LIN {X 0,Y 523.406,Z 267.821,A -85,B 0,C 180,E1 -4877.989,E2 -4877.989} C_VEL
LIN {X 0,Y 523.415,Z 265.36,A -85,B 0,C 180,E1 -4880.433,E2 -4880.433} C_VEL
LIN {X 0,Y 523.474,Z 262.881,A -85,B 0,C 180,E1 -4882.914,E2 -4882.914} C_VEL
LIN {X 0,Y 523.555,Z 259.879,A -85,B 0,C 180,E1 -4885.922,E2 -4885.922} C_VEL
LIN {X 0,Y 523.518,Z 256.912,A -85,B 0,C 180,E1 -4888.9,E2 -4888.9} C_VEL
LIN {X 0,Y 523.561,Z 255.036,A -85,B 0,C 180,E1 -4890.784,E2 -4890.784} C_VEL
LIN {X 0,Y 523.861,Z 254.859,A -85,B 0,C 180,E1 -4893.718,E2 -4893.718} C_VEL
LIN {X 0,Y 523.902,Z 254.849,A -85,B 0,C 180,E1 -4896.4,E2 -4896.4} C_VEL
LIN {X 0,Y 523.923,Z 254.848,A -85,B 0,C 180,E1 -4899.085,E2 -4899.085} C_VEL
LIN {X 0,Y 523.941,Z 254.846,A -85,B 0,C 180,E1 -4901.106,E2 -4901.106} C_VEL
LIN {X 0,Y 523.299,Z 254.928,A -85,B 0,C 180,E1 -4901.746,E2 -4901.746} C_VEL
LIN {X 0,Y 520.427,Z 255.284,A -85,B 0,C 180,E1 -4902.786,E2 -4902.786} C_VEL
LIN {X 0,Y 517.987,Z 255.586,A -85,B 0,C 180,E1 -4903.623,E2 -4903.623} C_VEL
LIN {X 0,Y 516.948,Z 255.716,A -85,B 0,C 180,E1 -4904.27,E2 -4904.27} C_VEL
LIN {X 0,Y 516.869,Z 255.723,A -85,B 0,C 180,E1 -4904.489,E2 -4904.489} C_VEL
LIN {X 0,Y 516.888,Z 255.725,A -85,B 0,C 180,E1 -4907.242,E2 -4907.242} C_VEL
LIN {X 0,Y 516.888,Z 255.725,A -85,B 0,C 180,E1 -4909.59,E2 -4909.59} C_VEL
LIN {X 0,Y 516.865,Z 255.729,A -85,B 0,C 180,E1 -4912.274,E2 -4912.274} C_VEL
LIN {X 0,Y 516.883,Z 255.728,A -85,B 0,C 180,E1 -4915.175,E2 -4915.175} C_VEL
LIN {X 0,Y 516.876,Z 255.725,A -85,B 0,C 180,E1 -4917.975,E2 -4917.975} C_VEL
LIN {X 0,Y 516.926,Z 255.719,A -85,B 0,C 180,E1 -4920.696,E2 -4920.696} C_VEL
LIN {X 0,Y 516.909,Z 255.722,A -85,B 0,C 180,E1 -4923.341,E2 -4923.341} C_VEL
LIN {X 0,Y 516.888,Z 255.726,A -85,B 0,C 180,E1 -4925.927,E2 -4925.927} C_VEL
LIN {X 0,Y 516.916,Z 255.722,A -85,B 0,C 180,E1 -4929.299,E2 -4929.299} C_VEL
LIN {X 0,Y 516.9,Z 255.723,A -85,B 0,C 180,E1 -4932.595,E2 -4932.595} C_VEL
LIN {X 0,Y 516.946,Z 255.72,A -85,B 0,C 180,E1 -4935.03,E2 -4935.03} C_VEL
LIN {X 0,Y 516.97,Z 255.718,A -85,B 0,C 180,E1 -4938.234,E2 -4938.234} C_VEL
LIN {X 0,Y 516.969,Z 255.717,A -85,B 0,C 180,E1 -4941.4,E2 -4941.4} C_VEL
LIN {X 0,Y 516.991,Z 255.712,A -85,B 0,C 180,E1 -4944.54,E2 -4944.54} C_VEL
LIN {X 0,Y 517.087,Z 255.701,A -85,B 0,C 180,E1 -4947.663,E2 -4947.663} C_VEL
LIN {X 0,Y 517.091,Z 255.699,A -85,B 0,C 180,E1 -4950.779,E2 -4950.779} C_VEL
LIN {X 0,Y 516.985,Z 255.713,A -85,B 0,C 180,E1 -4953.117,E2 -4953.117} C_VEL
LIN {X 0,Y 516.997,Z 255.713,A -85,B 0,C 180,E1 -4956.243,E2 -4956.243} C_VEL
LIN {X 0,Y 516.942,Z 255.719,A -85,B 0,C 180,E1 -4959.39,E2 -4959.39} C_VEL
LIN {X 0,Y 516.956,Z 255.715,A -85,B 0,C 180,E1 -4961.807,E2 -4961.807} C_VEL
LIN {X 0,Y 516.943,Z 255.717,A -85,B 0,C 180,E1 -4965.144,E2 -4965.144} C_VEL
LIN {X 0,Y 516.92,Z 255.721,A -85,B 0,C 180,E1 -4968.223,E2 -4968.223} C_VEL
LIN {X 0,Y 516.916,Z 255.72,A -85,B 0,C 180,E1 -4970.702,E2 -4970.702} C_VEL
LIN {X 0,Y 516.905,Z 255.721,A -85,B 0,C 180,E1 -4974.073,E2 -4974.073} C_VEL
LIN {X 0,Y 516.926,Z 255.72,A -85,B 0,C 180,E1 -4976.658,E2 -4976.658} C_VEL
LIN {X 0,Y 516.91,Z 255.723,A -85,B 0,C 180,E1 -4979.523,E2 -4979.523} C_VEL
LIN {X 0,Y 516.9,Z 255.726,A -85,B 0,C 180,E1 -4982.543,E2 -4982.543} C_VEL
LIN {X 0,Y 516.866,Z 255.731,A -85,B 0,C 180,E1 -4985.329,E2 -4985.329} C_VEL
LIN {X 0,Y 516.882,Z 255.725,A -85,B 0,C 180,E1 -4987.943,E2 -4987.943} C_VEL
LIN {X 0,Y 516.864,Z 255.727,A -85,B 0,C 180,E1 -4990.744,E2 -4990.744} C_VEL
LIN {X 0,Y 516.884,Z 255.723,A -85,B 0,C 180,E1 -4993.904,E2 -4993.904} C_VEL
LIN {X 0,Y 516.887,Z 255.727,A -85,B 0,C 180,E1 -4996.107,E2 -4996.107} C_VEL
LIN {X 0,Y 516.917,Z 255.72,A -85,B 0,C 180,E1 -4998.399,E2 -4998.399} C_VEL
LIN {X 0,Y 516.883,Z 255.724,A -85,B 0,C 180,E1 -5001.284,E2 -5001.284} C_VEL
LIN {X 0,Y 516.875,Z 255.726,A -85,B 0,C 180,E1 -5004.22,E2 -5004.22} C_VEL
LIN {X 0,Y 516.886,Z 255.725,A -85,B 0,C 180,E1 -5007.052,E2 -5007.052} C_VEL
LIN {X 0,Y 516.897,Z 255.725,A -85,B 0,C 180,E1 -5009.796,E2 -5009.796} C_VEL
LIN {X 0,Y 516.928,Z 255.72,A -85,B 0,C 180,E1 -5012.467,E2 -5012.467} C_VEL
LIN {X 0,Y 516.89,Z 255.725,A -85,B 0,C 180,E1 -5015.642,E2 -5015.642} C_VEL
LIN {X 0,Y 516.89,Z 255.724,A -85,B 0,C 180,E1 -5018.462,E2 -5018.462} C_VEL
LIN {X 0,Y 516.896,Z 255.722,A -85,B 0,C 180,E1 -5020.954,E2 -5020.954} C_VEL
LIN {X 0,Y 516.907,Z 255.724,A -85,B 0,C 180,E1 -5023.41,E2 -5023.41} C_VEL
LIN {X 0,Y 516.886,Z 255.724,A -85,B 0,C 180,E1 -5025.833,E2 -5025.833} C_VEL
LIN {X 0,Y 516.957,Z 255.715,A -85,B 0,C 180,E1 -5029.028,E2 -5029.028} C_VEL
LIN {X 0,Y 516.949,Z 255.717,A -85,B 0,C 180,E1 -5032.186,E2 -5032.186} C_VEL
LIN {X 0,Y 516.991,Z 255.711,A -85,B 0,C 180,E1 -5034.539,E2 -5034.539} C_VEL
LIN {X 0,Y 517.088,Z 255.7,A -85,B 0,C 180,E1 -5037.663,E2 -5037.663} C_VEL
LIN {X 0,Y 517.09,Z 255.701,A -85,B 0,C 180,E1 -5040,E2 -5040} C_VEL
LIN {X 0,Y 517.014,Z 255.71,A -85,B 0,C 180,E1 -5043.117,E2 -5043.117} C_VEL
LIN {X 0,Y 516.992,Z 255.715,A -85,B 0,C 180,E1 -5046.243,E2 -5046.243} C_VEL
LIN {X 0,Y 516.944,Z 255.72,A -85,B 0,C 180,E1 -5049.389,E2 -5049.389} C_VEL
LIN {X 0,Y 516.957,Z 255.716,A -85,B 0,C 180,E1 -5051.807,E2 -5051.807} C_VEL
LIN {X 0,Y 516.943,Z 255.717,A -85,B 0,C 180,E1 -5055.144,E2 -5055.144} C_VEL
LIN {X 0,Y 516.921,Z 255.722,A -85,B 0,C 180,E1 -5058.222,E2 -5058.222} C_VEL
LIN {X 0,Y 516.909,Z 255.72,A -85,B 0,C 180,E1 -5060.701,E2 -5060.701} C_VEL
LIN {X 0,Y 516.893,Z 255.724,A -85,B 0,C 180,E1 -5064.073,E2 -5064.073} C_VEL
LIN {X 0,Y 516.893,Z 255.723,A -85,B 0,C 180,E1 -5066.659,E2 -5066.659} C_VEL
LIN {X 0,Y 516.889,Z 255.725,A -85,B 0,C 180,E1 -5069.518,E2 -5069.518} C_VEL
LIN {X 0,Y 516.898,Z 255.724,A -85,B 0,C 180,E1 -5072.543,E2 -5072.543} C_VEL
LIN {X 0,Y 516.863,Z 255.73,A -85,B 0,C 180,E1 -5075.328,E2 -5075.328} C_VEL
LIN {X 0,Y 516.884,Z 255.725,A -85,B 0,C 180,E1 -5077.943,E2 -5077.943} C_VEL
LIN {X 0,Y 516.863,Z 255.727,A -85,B 0,C 180,E1 -5080.743,E2 -5080.743} C_VEL
LIN {X 0,Y 516.93,Z 255.935,A -85,B 0,C 180,E1 -5083.898,E2 -5083.898} C_VEL
LIN {X 0,Y 518.179,Z 262.543,A -85,B 0,C 180,E1 -5087.087,E2 -5087.087} C_VEL
LIN {X 0,Y 518.507,Z 266.609,A -85,B 0,C 180,E1 -5088.899,E2 -5088.899} C_VEL
LIN {X 0,Y 518.31,Z 272.634,A -85,B 0,C 180,E1 -5091.41,E2 -5091.41} C_VEL
LIN {X 0,Y 518.056,Z 279.916,A -85,B 0,C 180,E1 -5094.314,E2 -5094.314} C_VEL
LIN {X 0,Y 517.764,Z 287.94,A -85,B 0,C 180,E1 -5097.306,E2 -5097.306} C_VEL
LIN {X 0,Y 517.585,Z 296.354,A -85,B 0,C 180,E1 -5100.345,E2 -5100.345} C_VEL
LIN {X 0,Y 517.316,Z 305.881,A -85,B 0,C 180,E1 -5103.72,E2 -5103.72} C_VEL
LIN {X 0,Y 517.036,Z 314.769,A -85,B 0,C 180,E1 -5106.784,E2 -5106.784} C_VEL
LIN {X 0,Y 516.833,Z 323.591,A -85,B 0,C 180,E1 -5109.764,E2 -5109.764} C_VEL
LIN {X 0,Y 516.808,Z 325.424,A -85,B 0,C 180,E1 -5110.376,E2 -5110.376} C_VEL
LIN {X 0,Y 520.665,Z 341.342,A -85,B 0,C 180,E1 -5110.82,E2 -5110.82} C_VEL
LIN {X 0,Y 520.389,Z 357.008,A -85,B 0,C 180,E1 -5111.264,E2 -5111.264} C_VEL
LIN {X 0,Y 520.036,Z 371.091,A -85,B 0,C 180,E1 -5111.817,E2 -5111.817} C_VEL
LIN {X 0,Y 519.543,Z 384.386,A -85,B 0,C 180,E1 -5112.483,E2 -5112.483} C_VEL
LIN {X 0,Y 518.999,Z 398.66,A -85,B 0,C 180,E1 -5113.377,E2 -5113.377} C_VEL
LIN {X 0,Y 518.459,Z 411.744,A -85,B 0,C 180,E1 -5114.386,E2 -5114.386} C_VEL
LIN {X 0,Y 517.949,Z 423.365,A -85,B 0,C 180,E1 -5115.462,E2 -5115.462} C_VEL
LIN {X 0,Y 517.566,Z 434.168,A -85,B 0,C 180,E1 -5116.653,E2 -5116.653} C_VEL
LIN {X 0,Y 517.117,Z 444.315,A -85,B 0,C 180,E1 -5117.983,E2 -5117.983} C_VEL
LIN {X 0,Y 516.889,Z 453.439,A -85,B 0,C 180,E1 -5119.423,E2 -5119.423} C_VEL
LIN {X 0,Y 516.581,Z 461.637,A -85,B 0,C 180,E1 -5120.999,E2 -5120.999} C_VEL
LIN {X 0,Y 516.428,Z 468.204,A -85,B 0,C 180,E1 -5122.572,E2 -5122.572} C_VEL
LIN {X 0,Y 516.378,Z 473.338,A -85,B 0,C 180,E1 -5124.141,E2 -5124.141} C_VEL
LIN {X 0,Y 516.239,Z 476.297,A -85,B 0,C 180,E1 -5125.315,E2 -5125.315} C_VEL
LIN {X 0,Y 516.271,Z 479.191,A -85,B 0,C 180,E1 -5126.879,E2 -5126.879} C_VEL
LIN {X 0,Y 516.189,Z 480.915,A -85,B 0,C 180,E1 -5128.44,E2 -5128.44} C_VEL
LIN {X 0,Y 516.151,Z 481.5,A -85,B 0,C 180,E1 -5130,E2 -5130} C_VEL
LIN {X 0,Y 516.189,Z 480.912,A -85,B 0,C 180,E1 -5131.56,E2 -5131.56} C_VEL
LIN {X 0,Y 516.271,Z 479.185,A -85,B 0,C 180,E1 -5133.121,E2 -5133.121} C_VEL
LIN {X 0,Y 516.239,Z 476.294,A -85,B 0,C 180,E1 -5134.685,E2 -5134.685} C_VEL
LIN {X 0,Y 516.376,Z 472.164,A -85,B 0,C 180,E1 -5136.251,E2 -5136.251} C_VEL
LIN {X 0,Y 516.463,Z 466.693,A -85,B 0,C 180,E1 -5137.821,E2 -5137.821} C_VEL
LIN {X 0,Y 516.627,Z 459.735,A -85,B 0,C 180,E1 -5139.395,E2 -5139.395} C_VEL
LIN {X 0,Y 516.974,Z 451.086,A -85,B 0,C 180,E1 -5140.972,E2 -5140.972} C_VEL
LIN {X 0,Y 517.204,Z 442.012,A -85,B 0,C 180,E1 -5142.338,E2 -5142.338} C_VEL
LIN {X 0,Y 517.611,Z 432.477,A -85,B 0,C 180,E1 -5143.546,E2 -5143.546} C_VEL
LIN {X 0,Y 518.043,Z 421.354,A -85,B 0,C 180,E1 -5144.736,E2 -5144.736} C_VEL
LIN {X 0,Y 518.503,Z 409.888,A -85,B 0,C 180,E1 -5145.77,E2 -5145.77} C_VEL
LIN {X 0,Y 519.031,Z 397.214,A -85,B 0,C 180,E1 -5146.723,E2 -5146.723} C_VEL
LIN {X 0,Y 519.558,Z 384.408,A -85,B 0,C 180,E1 -5147.516,E2 -5147.516} C_VEL
LIN {X 0,Y 520.032,Z 371.116,A -85,B 0,C 180,E1 -5148.183,E2 -5148.183} C_VEL
LIN {X 0,Y 520.461,Z 355.507,A -85,B 0,C 180,E1 -5148.785,E2 -5148.785} C_VEL
LIN {X 0,Y 520.675,Z 341.247,A -85,B 0,C 180,E1 -5149.183,E2 -5149.183} C_VEL
LIN {X 0,Y 516.802,Z 325.427,A -85,B 0,C 180,E1 -5149.623,E2 -5149.623} C_VEL
LIN {X 0,Y 516.961,Z 318.483,A -85,B 0,C 180,E1 -5151.954,E2 -5151.954} C_VEL
LIN {X 0,Y 517.153,Z 309.818,A -85,B 0,C 180,E1 -5154.916,E2 -5154.916} C_VEL
LIN {X 0,Y 517.345,Z 302.391,A -85,B 0,C 180,E1 -5157.509,E2 -5157.509} C_VEL
LIN {X 0,Y 517.567,Z 294.891,A -85,B 0,C 180,E1 -5160.16,E2 -5160.16} C_VEL
LIN {X 0,Y 517.732,Z 285.622,A -85,B 0,C 180,E1 -5163.352,E2 -5163.352} C_VEL
LIN {X 0,Y 517.912,Z 279.176,A -85,B 0,C 180,E1 -5165.698,E2 -5165.698} C_VEL
LIN {X 0,Y 518.22,Z 272.13,A -85,B 0,C 180,E1 -5168.598,E2 -5168.598} C_VEL
LIN {X 0,Y 518.476,Z 267.989,A -85,B 0,C 180,E1 -5170.616,E2 -5170.616} C_VEL
LIN {X 0,Y 518.547,Z 265.926,A -85,B 0,C 180,E1 -5171.804,E2 -5171.804} C_VEL
LIN {X 0,Y 518.255,Z 263.34,A -85,B 0,C 180,E1 -5173.758,E2 -5173.758} C_VEL
LIN {X 0,Y 517.9,Z 261.592,A -85,B 0,C 180,E1 -5175.991,E2 -5175.991} C_VEL
LIN {X 0,Y 517.599,Z 261.084,A -85,B 0,C 180,E1 -5178.314,E2 -5178.314} C_VEL
LIN {X 0,Y 517.206,Z 261.849,A -85,B 0,C 180,E1 -5181.313,E2 -5181.313} C_VEL
LIN {X 0,Y 516.978,Z 263.353,A -85,B 0,C 180,E1 -5184.228,E2 -5184.228} C_VEL
LIN {X 0,Y 516.825,Z 265.149,A -85,B 0,C 180,E1 -5187.048,E2 -5187.048} C_VEL
LIN {X 0,Y 516.727,Z 267.071,A -85,B 0,C 180,E1 -5189.786,E2 -5189.786} C_VEL
LIN {X 0,Y 516.626,Z 269.077,A -85,B 0,C 180,E1 -5192.45,E2 -5192.45} C_VEL
LIN {X 0,Y 516.508,Z 271.145,A -85,B 0,C 180,E1 -5195.051,E2 -5195.051} C_VEL
LIN {X 0,Y 516.464,Z 272.453,A -85,B 0,C 180,E1 -5196.638,E2 -5196.638} C_VEL
LIN {X 0,Y 520.318,Z 286.354,A -85,B 0,C 180,E1 -5197.076,E2 -5197.076} C_VEL
LIN {X 0,Y 520.049,Z 302.179,A -85,B 0,C 180,E1 -5197.565,E2 -5197.565} C_VEL
LIN {X 0,Y 519.665,Z 317.564,A -85,B 0,C 180,E1 -5198.219,E2 -5198.219} C_VEL
LIN {X 0,Y 519.183,Z 331.854,A -85,B 0,C 180,E1 -5199,E2 -5199} C_VEL
LIN {X 0,Y 518.738,Z 345.039,A -85,B 0,C 180,E1 -5199.892,E2 -5199.892} C_VEL
LIN {X 0,Y 518.269,Z 357.321,A -85,B 0,C 180,E1 -5200.904,E2 -5200.904} C_VEL
LIN {X 0,Y 517.822,Z 369.228,A -85,B 0,C 180,E1 -5202.082,E2 -5202.082} C_VEL
LIN {X 0,Y 517.375,Z 380.417,A -85,B 0,C 180,E1 -5203.426,E2 -5203.426} C_VEL
LIN {X 0,Y 517.06,Z 388.916,A -85,B 0,C 180,E1 -5204.64,E2 -5204.64} C_VEL
LIN {X 0,Y 516.787,Z 397.101,A -85,B 0,C 180,E1 -5206.032,E2 -5206.032} C_VEL
LIN {X 0,Y 516.568,Z 403.816,A -85,B 0,C 180,E1 -5207.427,E2 -5207.427} C_VEL
LIN {X 0,Y 516.41,Z 410.046,A -85,B 0,C 180,E1 -5209.016,E2 -5209.016} C_VEL
LIN {X 0,Y 516.275,Z 414.768,A -85,B 0,C 180,E1 -5210.599,E2 -5210.599} C_VEL
LIN {X 0,Y 516.26,Z 418.206,A -85,B 0,C 180,E1 -5212.176,E2 -5212.176} C_VEL
LIN {X 0,Y 516.295,Z 420.481,A -85,B 0,C 180,E1 -5213.748,E2 -5213.748} C_VEL
LIN {X 0,Y 516.213,Z 421.519,A -85,B 0,C 180,E1 -5215.315,E2 -5215.315} C_VEL
LIN {X 0,Y 516.278,Z 421.689,A -85,B 0,C 180,E1 -5216.097,E2 -5216.097} C_VEL
LIN {X 0,Y 516.258,Z 421.036,A -85,B 0,C 180,E1 -5217.66,E2 -5217.66} C_VEL
LIN {X 0,Y 516.16,Z 419.321,A -85,B 0,C 180,E1 -5219.22,E2 -5219.22} C_VEL
LIN {X 0,Y 516.181,Z 416.483,A -85,B 0,C 180,E1 -5220.78,E2 -5220.78} C_VEL
LIN {X 0,Y 516.314,Z 412.311,A -85,B 0,C 180,E1 -5222.341,E2 -5222.341} C_VEL
LIN {X 0,Y 516.495,Z 408.36,A -85,B 0,C 180,E1 -5223.511,E2 -5223.511} C_VEL
LIN {X 0,Y 516.663,Z 401.892,A -85,B 0,C 180,E1 -5225.073,E2 -5225.073} C_VEL
LIN {X 0,Y 516.849,Z 394.528,A -85,B 0,C 180,E1 -5226.5,E2 -5226.5} C_VEL
LIN {X 0,Y 517.127,Z 386.378,A -85,B 0,C 180,E1 -5227.811,E2 -5227.811} C_VEL
LIN {X 0,Y 517.527,Z 376.249,A -85,B 0,C 180,E1 -5229.182,E2 -5229.182} C_VEL
LIN {X 0,Y 517.917,Z 365.769,A -85,B 0,C 180,E1 -5230.358,E2 -5230.358} C_VEL
LIN {X 0,Y 518.424,Z 354.456,A -85,B 0,C 180,E1 -5231.436,E2 -5231.436} C_VEL
LIN {X 0,Y 518.943,Z 340.7,A -85,B 0,C 180,E1 -5232.515,E2 -5232.515} C_VEL
LIN {X 0,Y 519.352,Z 328.639,A -85,B 0,C 180,E1 -5233.3,E2 -5233.3} C_VEL
LIN {X 0,Y 519.838,Z 313.549,A -85,B 0,C 180,E1 -5234.085,E2 -5234.085} C_VEL
LIN {X 0,Y 520.268,Z 298.968,A -85,B 0,C 180,E1 -5234.672,E2 -5234.672} C_VEL
LIN {X 0,Y 520.386,Z 286.11,A -85,B 0,C 180,E1 -5235.065,E2 -5235.065} C_VEL
LIN {X 0,Y 516.998,Z 273.328,A -85,B 0,C 180,E1 -5235.464,E2 -5235.464} C_VEL
LIN {X 0,Y 516.35,Z 270.85,A -85,B 0,C 180,E1 -5235.555,E2 -5235.555} C_VEL
LIN {X 0,Y 516.342,Z 268.172,A -85,B 0,C 180,E1 -5238.244,E2 -5238.244} C_VEL
LIN {X 0,Y 516.353,Z 265.672,A -85,B 0,C 180,E1 -5240.725,E2 -5240.725} C_VEL
LIN {X 0,Y 516.424,Z 263.167,A -85,B 0,C 180,E1 -5243.245,E2 -5243.245} C_VEL
LIN {X 0,Y 516.487,Z 260.344,A -85,B 0,C 180,E1 -5246.092,E2 -5246.092} C_VEL
LIN {X 0,Y 516.435,Z 258.002,A -85,B 0,C 180,E1 -5248.445,E2 -5248.445} C_VEL
LIN {X 0,Y 516.461,Z 256.231,A -85,B 0,C 180,E1 -5250.232,E2 -5250.232} C_VEL
LIN {X 0,Y 516.523,Z 255.774,A -85,B 0,C 180,E1 -5251.134,E2 -5251.134} C_VEL
LIN {X 0,Y 516.82,Z 255.735,A -85,B 0,C 180,E1 -5253.951,E2 -5253.951} C_VEL
LIN {X 0,Y 516.857,Z 255.728,A -85,B 0,C 180,E1 -5256.748,E2 -5256.748} C_VEL
LIN {X 0,Y 516.886,Z 255.725,A -85,B 0,C 180,E1 -5259.721,E2 -5259.721} C_VEL
LIN {X 0,Y 516.909,Z 255.723,A -85,B 0,C 180,E1 -5261.776,E2 -5261.776} C_VEL
LIN {X 0,Y 516.869,Z 255.723,A -85,B 0,C 180,E1 -5264.489,E2 -5264.489} C_VEL
LIN {X 0,Y 516.212,Z 255.809,A -85,B 0,C 180,E1 -5265.14,E2 -5265.14} C_VEL
LIN {X 0,Y 513.347,Z 256.167,A -85,B 0,C 180,E1 -5266.196,E2 -5266.196} C_VEL
LIN {X 0,Y 510.932,Z 256.468,A -85,B 0,C 180,E1 -5267.046,E2 -5267.046} C_VEL
LIN {X 0,Y 509.917,Z 256.595,A -85,B 0,C 180,E1 -5267.704,E2 -5267.704} C_VEL
LIN {X 0,Y 509.847,Z 256.602,A -85,B 0,C 180,E1 -5267.926,E2 -5267.926} C_VEL
LIN {X 0,Y 509.848,Z 256.603,A -85,B 0,C 180,E1 -5270.647,E2 -5270.647} C_VEL
LIN {X 0,Y 509.828,Z 256.606,A -85,B 0,C 180,E1 -5273.647,E2 -5273.647} C_VEL
LIN {X 0,Y 509.845,Z 256.602,A -85,B 0,C 180,E1 -5276.538,E2 -5276.538} C_VEL
LIN {X 0,Y 509.849,Z 256.601,A -85,B 0,C 180,E1 -5279.334,E2 -5279.334} C_VEL
LIN {X 0,Y 509.895,Z 256.595,A -85,B 0,C 180,E1 -5282.054,E2 -5282.054} C_VEL
LIN {X 0,Y 509.811,Z 256.607,A -85,B 0,C 180,E1 -5284.7,E2 -5284.7} C_VEL
LIN {X 0,Y 509.83,Z 256.605,A -85,B 0,C 180,E1 -5287.458,E2 -5287.458} C_VEL
LIN {X 0,Y 509.92,Z 256.591,A -85,B 0,C 180,E1 -5289.845,E2 -5289.845} C_VEL
LIN {X 0,Y 509.872,Z 256.598,A -85,B 0,C 180,E1 -5293.174,E2 -5293.174} C_VEL
LIN {X 0,Y 509.863,Z 256.6,A -85,B 0,C 180,E1 -5295.634,E2 -5295.634} C_VEL
LIN {X 0,Y 509.916,Z 256.591,A -85,B 0,C 180,E1 -5298.875,E2 -5298.875} C_VEL
LIN {X 0,Y 509.955,Z 256.588,A -85,B 0,C 180,E1 -5302.078,E2 -5302.078} C_VEL
LIN {X 0,Y 509.946,Z 256.59,A -85,B 0,C 180,E1 -5304.464,E2 -5304.464} C_VEL
LIN {X 0,Y 510.056,Z 256.577,A -85,B 0,C 180,E1 -5307.631,E2 -5307.631} C_VEL
LIN {X 0,Y 510.06,Z 256.576,A -85,B 0,C 180,E1 -5310,E2 -5310} C_VEL
LIN {X 0,Y 510.053,Z 256.575,A -85,B 0,C 180,E1 -5312.369,E2 -5312.369} C_VEL
LIN {X 0,Y 509.979,Z 256.585,A -85,B 0,C 180,E1 -5315.536,E2 -5315.536} C_VEL
LIN {X 0,Y 509.905,Z 256.592,A -85,B 0,C 180,E1 -5318.72,E2 -5318.72} C_VEL
LIN {X 0,Y 509.908,Z 256.594,A -85,B 0,C 180,E1 -5321.932,E2 -5321.932} C_VEL
LIN {X 0,Y 509.898,Z 256.595,A -85,B 0,C 180,E1 -5325.242,E2 -5325.242} C_VEL
LIN {X 0,Y 509.865,Z 256.601,A -85,B 0,C 180,E1 -5328.484,E2 -5328.484} C_VEL
LIN {X 0,Y 509.854,Z 256.6,A -85,B 0,C 180,E1 -5331.002,E2 -5331.002} C_VEL
LIN {X 0,Y 509.867,Z 256.6,A -85,B 0,C 180,E1 -5334.426,E2 -5334.426} C_VEL
LIN {X 0,Y 509.884,Z 256.596,A -85,B 0,C 180,E1 -5337.056,E2 -5337.056} C_VEL
LIN {X 0,Y 509.86,Z 256.599,A -85,B 0,C 180,E1 -5339.751,E2 -5339.751} C_VEL
LIN {X 0,Y 509.877,Z 256.598,A -85,B 0,C 180,E1 -5342.774,E2 -5342.774} C_VEL
LIN {X 0,Y 509.826,Z 256.605,A -85,B 0,C 180,E1 -5345.578,E2 -5345.578} C_VEL
LIN {X 0,Y 509.853,Z 256.602,A -85,B 0,C 180,E1 -5348.338,E2 -5348.338} C_VEL
LIN {X 0,Y 509.812,Z 256.609,A -85,B 0,C 180,E1 -5351.43,E2 -5351.43} C_VEL
LIN {X 0,Y 509.843,Z 256.605,A -85,B 0,C 180,E1 -5354.67,E2 -5354.67} C_VEL
LIN {X 0,Y 509.838,Z 256.605,A -85,B 0,C 180,E1 -5357.51,E2 -5357.51} C_VEL
LIN {X 0,Y 509.849,Z 256.605,A -85,B 0,C 180,E1 -5360.647,E2 -5360.647} C_VEL
LIN {X 0,Y 509.829,Z 256.606,A -85,B 0,C 180,E1 -5363.647,E2 -5363.647} C_VEL
LIN {X 0,Y 509.846,Z 256.603,A -85,B 0,C 180,E1 -5366.538,E2 -5366.538} C_VEL
LIN {X 0,Y 509.85,Z 256.602,A -85,B 0,C 180,E1 -5369.334,E2 -5369.334} C_VEL
LIN {X 0,Y 509.895,Z 256.594,A -85,B 0,C 180,E1 -5372.054,E2 -5372.054} C_VEL
LIN {X 0,Y 509.829,Z 256.604,A -85,B 0,C 180,E1 -5374.701,E2 -5374.701} C_VEL
LIN {X 0,Y 509.832,Z 256.605,A -85,B 0,C 180,E1 -5377.458,E2 -5377.458} C_VEL
LIN {X 0,Y 509.92,Z 256.591,A -85,B 0,C 180,E1 -5379.845,E2 -5379.845} C_VEL
LIN {X 0,Y 509.873,Z 256.6,A -85,B 0,C 180,E1 -5383.174,E2 -5383.174} C_VEL
LIN {X 0,Y 509.858,Z 256.599,A -85,B 0,C 180,E1 -5385.634,E2 -5385.634} C_VEL
LIN {X 0,Y 509.919,Z 256.592,A -85,B 0,C 180,E1 -5388.874,E2 -5388.874} C_VEL
LIN {X 0,Y 509.914,Z 256.593,A -85,B 0,C 180,E1 -5392.078,E2 -5392.078} C_VEL
LIN {X 0,Y 509.946,Z 256.589,A -85,B 0,C 180,E1 -5394.464,E2 -5394.464} C_VEL
LIN {X 0,Y 510.057,Z 256.576,A -85,B 0,C 180,E1 -5397.631,E2 -5397.631} C_VEL
LIN {X 0,Y 510.061,Z 256.577,A -85,B 0,C 180,E1 -5400,E2 -5400} C_VEL
LIN {X 0,Y 510.059,Z 256.574,A -85,B 0,C 180,E1 -5402.369,E2 -5402.369} C_VEL
LIN {X 0,Y 509.978,Z 256.585,A -85,B 0,C 180,E1 -5405.536,E2 -5405.536} C_VEL
LIN {X 0,Y 509.89,Z 256.595,A -85,B 0,C 180,E1 -5408.72,E2 -5408.72} C_VEL
LIN {X 0,Y 509.909,Z 256.594,A -85,B 0,C 180,E1 -5411.931,E2 -5411.931} C_VEL
LIN {X 0,Y 509.899,Z 256.596,A -85,B 0,C 180,E1 -5415.241,E2 -5415.241} C_VEL
LIN {X 0,Y 509.866,Z 256.601,A -85,B 0,C 180,E1 -5418.483,E2 -5418.483} C_VEL
LIN {X 0,Y 509.85,Z 256.6,A -85,B 0,C 180,E1 -5421.002,E2 -5421.002} C_VEL
LIN {X 0,Y 509.824,Z 256.604,A -85,B 0,C 180,E1 -5423.564,E2 -5423.564} C_VEL
LIN {X 0,Y 509.878,Z 256.599,A -85,B 0,C 180,E1 -5426.37,E2 -5426.37} C_VEL
LIN {X 0,Y 509.854,Z 256.6,A -85,B 0,C 180,E1 -5429.751,E2 -5429.751} C_VEL
LIN {X 0,Y 509.873,Z 256.598,A -85,B 0,C 180,E1 -5432.773,E2 -5432.773} C_VEL
LIN {X 0,Y 509.824,Z 256.605,A -85,B 0,C 180,E1 -5435.577,E2 -5435.577} C_VEL
LIN {X 0,Y 509.853,Z 256.601,A -85,B 0,C 180,E1 -5438.338,E2 -5438.338} C_VEL
LIN {X 0,Y 509.834,Z 256.605,A -85,B 0,C 180,E1 -5441.427,E2 -5441.427} C_VEL
LIN {X 0,Y 509.841,Z 256.716,A -85,B 0,C 180,E1 -5443.424,E2 -5443.424} C_VEL
LIN {X 0,Y 511.063,Z 263.043,A -85,B 0,C 180,E1 -5446.56,E2 -5446.56} C_VEL
LIN {X 0,Y 511.51,Z 265.916,A -85,B 0,C 180,E1 -5447.897,E2 -5447.897} C_VEL
LIN {X 0,Y 511.484,Z 271.465,A -85,B 0,C 180,E1 -5450.306,E2 -5450.306} C_VEL
LIN {X 0,Y 511.202,Z 278.822,A -85,B 0,C 180,E1 -5453.319,E2 -5453.319} C_VEL
LIN {X 0,Y 510.881,Z 286.102,A -85,B 0,C 180,E1 -5456.141,E2 -5456.141} C_VEL
LIN {X 0,Y 510.607,Z 294.884,A -85,B 0,C 180,E1 -5459.385,E2 -5459.385} C_VEL
LIN {X 0,Y 510.39,Z 302.391,A -85,B 0,C 180,E1 -5462.084,E2 -5462.084} C_VEL
LIN {X 0,Y 510.157,Z 309.818,A -85,B 0,C 180,E1 -5464.719,E2 -5464.719} C_VEL
LIN {X 0,Y 509.937,Z 318.662,A -85,B 0,C 180,E1 -5467.789,E2 -5467.789} C_VEL
LIN {X 0,Y 509.769,Z 325.428,A -85,B 0,C 180,E1 -5470.095,E2 -5470.095} C_VEL
LIN {X 0,Y 513.784,Z 341.933,A -85,B 0,C 180,E1 -5470.567,E2 -5470.567} C_VEL
LIN {X 0,Y 513.969,Z 347.826,A -85,B 0,C 180,E1 -5470.73,E2 -5470.73} C_VEL
LIN {X 0,Y 513.534,Z 362.77,A -85,B 0,C 180,E1 -5471.222,E2 -5471.222} C_VEL
LIN {X 0,Y 512.994,Z 377.835,A -85,B 0,C 180,E1 -5471.891,E2 -5471.891} C_VEL
LIN {X 0,Y 512.49,Z 391.111,A -85,B 0,C 180,E1 -5472.646,E2 -5472.646} C_VEL
LIN {X 0,Y 511.947,Z 404.102,A -85,B 0,C 180,E1 -5473.552,E2 -5473.552} C_VEL
LIN {X 0,Y 511.422,Z 415.612,A -85,B 0,C 180,E1 -5474.515,E2 -5474.515} C_VEL
LIN {X 0,Y 510.888,Z 427.155,A -85,B 0,C 180,E1 -5475.663,E2 -5475.663} C_VEL
LIN {X 0,Y 510.419,Z 437.363,A -85,B 0,C 180,E1 -5476.868,E2 -5476.868} C_VEL
LIN {X 0,Y 509.987,Z 447.098,A -85,B 0,C 180,E1 -5478.234,E2 -5478.234} C_VEL
LIN {X 0,Y 509.745,Z 455.642,A -85,B 0,C 180,E1 -5479.675,E2 -5479.675} C_VEL
LIN {X 0,Y 509.482,Z 463.412,A -85,B 0,C 180,E1 -5481.272,E2 -5481.272} C_VEL
LIN {X 0,Y 509.318,Z 469.602,A -85,B 0,C 180,E1 -5482.866,E2 -5482.866} C_VEL
LIN {X 0,Y 509.284,Z 474.389,A -85,B 0,C 180,E1 -5484.457,E2 -5484.457} C_VEL
LIN {X 0,Y 509.201,Z 477.895,A -85,B 0,C 180,E1 -5486.043,E2 -5486.043} C_VEL
LIN {X 0,Y 509.158,Z 480.196,A -85,B 0,C 180,E1 -5487.627,E2 -5487.627} C_VEL
LIN {X 0,Y 509.07,Z 481.351,A -85,B 0,C 180,E1 -5489.209,E2 -5489.209} C_VEL
LIN {X 0,Y 509.07,Z 481.35,A -85,B 0,C 180,E1 -5490.791,E2 -5490.791} C_VEL
LIN {X 0,Y 509.158,Z 480.191,A -85,B 0,C 180,E1 -5492.373,E2 -5492.373} C_VEL
LIN {X 0,Y 509.201,Z 477.889,A -85,B 0,C 180,E1 -5493.957,E2 -5493.957} C_VEL
LIN {X 0,Y 509.285,Z 474.388,A -85,B 0,C 180,E1 -5495.543,E2 -5495.543} C_VEL
LIN {X 0,Y 509.32,Z 469.603,A -85,B 0,C 180,E1 -5497.134,E2 -5497.134} C_VEL
LIN {X 0,Y 509.481,Z 463.409,A -85,B 0,C 180,E1 -5498.728,E2 -5498.728} C_VEL
LIN {X 0,Y 509.745,Z 455.636,A -85,B 0,C 180,E1 -5500.325,E2 -5500.325} C_VEL
LIN {X 0,Y 510.009,Z 447.014,A -85,B 0,C 180,E1 -5501.778,E2 -5501.778} C_VEL
LIN {X 0,Y 510.419,Z 437.361,A -85,B 0,C 180,E1 -5503.132,E2 -5503.132} C_VEL
LIN {X 0,Y 510.868,Z 427.158,A -85,B 0,C 180,E1 -5504.337,E2 -5504.337} C_VEL
LIN {X 0,Y 511.408,Z 415.77,A -85,B 0,C 180,E1 -5505.471,E2 -5505.471} C_VEL
LIN {X 0,Y 511.934,Z 404.124,A -85,B 0,C 180,E1 -5506.448,E2 -5506.448} C_VEL
LIN {X 0,Y 512.464,Z 391.13,A -85,B 0,C 180,E1 -5507.355,E2 -5507.355} C_VEL
LIN {X 0,Y 513.037,Z 376.841,A -85,B 0,C 180,E1 -5508.159,E2 -5508.159} C_VEL
LIN {X 0,Y 513.571,Z 362.82,A -85,B 0,C 180,E1 -5508.777,E2 -5508.777} C_VEL
LIN {X 0,Y 513.918,Z 347.951,A -85,B 0,C 180,E1 -5509.27,E2 -5509.27} C_VEL
LIN {X 0,Y 513.947,Z 342.538,A -85,B 0,C 180,E1 -5509.415,E2 -5509.415} C_VEL
LIN {X 0,Y 509.876,Z 326.129,A -85,B 0,C 180,E1 -5509.889,E2 -5509.889} C_VEL
LIN {X 0,Y 509.772,Z 325.352,A -85,B 0,C 180,E1 -5509.93,E2 -5509.93} C_VEL
LIN {X 0,Y 509.958,Z 317.245,A -85,B 0,C 180,E1 -5512.699,E2 -5512.699} C_VEL
LIN {X 0,Y 510.198,Z 308.58,A -85,B 0,C 180,E1 -5515.716,E2 -5515.716} C_VEL
LIN {X 0,Y 510.495,Z 299.795,A -85,B 0,C 180,E1 -5518.806,E2 -5518.806} C_VEL
LIN {X 0,Y 510.614,Z 290.493,A -85,B 0,C 180,E1 -5521.999,E2 -5521.999} C_VEL
LIN {X 0,Y 510.864,Z 282.664,A -85,B 0,C 180,E1 -5524.814,E2 -5524.814} C_VEL
LIN {X 0,Y 511.131,Z 275.462,A -85,B 0,C 180,E1 -5527.725,E2 -5527.725} C_VEL
LIN {X 0,Y 511.45,Z 270.185,A -85,B 0,C 180,E1 -5530.229,E2 -5530.229} C_VEL
LIN {X 0,Y 511.55,Z 266.695,A -85,B 0,C 180,E1 -5532.314,E2 -5532.314} C_VEL
LIN {X 0,Y 511.171,Z 264.159,A -85,B 0,C 180,E1 -5534.523,E2 -5534.523} C_VEL
LIN {X 0,Y 510.852,Z 262.767,A -85,B 0,C 180,E1 -5536.815,E2 -5536.815} C_VEL
LIN {X 0,Y 510.473,Z 262.573,A -85,B 0,C 180,E1 -5539.22,E2 -5539.22} C_VEL
LIN {X 0,Y 510.167,Z 263.285,A -85,B 0,C 180,E1 -5541.742,E2 -5541.742} C_VEL
LIN {X 0,Y 509.942,Z 264.714,A -85,B 0,C 180,E1 -5544.631,E2 -5544.631} C_VEL
LIN {X 0,Y 509.788,Z 266.487,A -85,B 0,C 180,E1 -5547.476,E2 -5547.476} C_VEL
LIN {X 0,Y 509.676,Z 268.448,A -85,B 0,C 180,E1 -5550.311,E2 -5550.311} C_VEL
LIN {X 0,Y 509.547,Z 270.391,A -85,B 0,C 180,E1 -5552.925,E2 -5552.925} C_VEL
LIN {X 0,Y 509.476,Z 272.818,A -85,B 0,C 180,E1 -5555.987,E2 -5555.987} C_VEL
LIN {X 0,Y 509.464,Z 273.388,A -85,B 0,C 180,E1 -5556.419,E2 -5556.419} C_VEL
LIN {X 0,Y 513.295,Z 286.754,A -85,B 0,C 180,E1 -5556.846,E2 -5556.846} C_VEL
LIN {X 0,Y 513.581,Z 289.783,A -85,B 0,C 180,E1 -5556.942,E2 -5556.942} C_VEL
LIN {X 0,Y 513.202,Z 304.185,A -85,B 0,C 180,E1 -5557.412,E2 -5557.412} C_VEL
LIN {X 0,Y 512.765,Z 319.13,A -85,B 0,C 180,E1 -5558.069,E2 -5558.069} C_VEL
LIN {X 0,Y 512.341,Z 331.893,A -85,B 0,C 180,E1 -5558.777,E2 -5558.777} C_VEL
LIN {X 0,Y 511.852,Z 345.596,A -85,B 0,C 180,E1 -5559.715,E2 -5559.715} C_VEL
LIN {X 0,Y 511.349,Z 357.919,A -85,B 0,C 180,E1 -5560.74,E2 -5560.74} C_VEL
LIN {X 0,Y 510.888,Z 369.558,A -85,B 0,C 180,E1 -5561.905,E2 -5561.905} C_VEL
LIN {X 0,Y 510.429,Z 380.275,A -85,B 0,C 180,E1 -5563.193,E2 -5563.193} C_VEL
LIN {X 0,Y 510.094,Z 388.828,A -85,B 0,C 180,E1 -5564.416,E2 -5564.416} C_VEL
LIN {X 0,Y 509.791,Z 397.171,A -85,B 0,C 180,E1 -5565.836,E2 -5565.836} C_VEL
LIN {X 0,Y 509.54,Z 404.008,A -85,B 0,C 180,E1 -5567.251,E2 -5567.251} C_VEL
LIN {X 0,Y 509.36,Z 410.285,A -85,B 0,C 180,E1 -5568.862,E2 -5568.862} C_VEL
LIN {X 0,Y 509.215,Z 415.113,A -85,B 0,C 180,E1 -5570.467,E2 -5570.467} C_VEL
LIN {X 0,Y 509.198,Z 418.588,A -85,B 0,C 180,E1 -5572.067,E2 -5572.067} C_VEL
LIN {X 0,Y 509.221,Z 420.898,A -85,B 0,C 180,E1 -5573.661,E2 -5573.661} C_VEL
LIN {X 0,Y 509.132,Z 421.992,A -85,B 0,C 180,E1 -5575.249,E2 -5575.249} C_VEL
LIN {X 0,Y 509.208,Z 422.164,A -85,B 0,C 180,E1 -5576.043,E2 -5576.043} C_VEL
LIN {X 0,Y 509.186,Z 421.552,A -85,B 0,C 180,E1 -5577.627,E2 -5577.627} C_VEL
LIN {X 0,Y 509.079,Z 419.851,A -85,B 0,C 180,E1 -5579.209,E2 -5579.209} C_VEL
LIN {X 0,Y 509.102,Z 417.016,A -85,B 0,C 180,E1 -5580.791,E2 -5580.791} C_VEL
LIN {X 0,Y 509.244,Z 412.876,A -85,B 0,C 180,E1 -5582.373,E2 -5582.373} C_VEL
LIN {X 0,Y 509.482,Z 407.473,A -85,B 0,C 180,E1 -5583.955,E2 -5583.955} C_VEL
LIN {X 0,Y 509.619,Z 400.592,A -85,B 0,C 180,E1 -5585.54,E2 -5585.54} C_VEL
LIN {X 0,Y 509.884,Z 393.956,A -85,B 0,C 180,E1 -5586.793,E2 -5586.793} C_VEL
LIN {X 0,Y 510.178,Z 385.667,A -85,B 0,C 180,E1 -5588.117,E2 -5588.117} C_VEL
LIN {X 0,Y 510.677,Z 375.248,A -85,B 0,C 180,E1 -5589.506,E2 -5589.506} C_VEL
LIN {X 0,Y 511.099,Z 364.509,A -85,B 0,C 180,E1 -5590.698,E2 -5590.698} C_VEL
LIN {X 0,Y 511.635,Z 351.689,A -85,B 0,C 180,E1 -5591.891,E2 -5591.891} C_VEL
LIN {X 0,Y 512.177,Z 338.621,A -85,B 0,C 180,E1 -5592.887,E2 -5592.887} C_VEL
LIN {X 0,Y 512.709,Z 324.314,A -85,B 0,C 180,E1 -5593.779,E2 -5593.779} C_VEL
LIN {X 0,Y 513.161,Z 310.172,A -85,B 0,C 180,E1 -5594.474,E2 -5594.474} C_VEL
LIN {X 0,Y 513.585,Z 295.084,A -85,B 0,C 180,E1 -5595.045,E2 -5595.045} C_VEL
LIN {X 0,Y 513.512,Z 286.851,A -85,B 0,C 180,E1 -5595.296,E2 -5595.296} C_VEL
LIN {X 0,Y 509.891,Z 273.663,A -85,B 0,C 180,E1 -5595.724,E2 -5595.724} C_VEL
LIN {X 0,Y 509.275,Z 271.243,A -85,B 0,C 180,E1 -5595.808,E2 -5595.808} C_VEL
LIN {X 0,Y 509.274,Z 268.527,A -85,B 0,C 180,E1 -5598.506,E2 -5598.506} C_VEL
LIN {X 0,Y 509.276,Z 265.988,A -85,B 0,C 180,E1 -5601.027,E2 -5601.027} C_VEL
LIN {X 0,Y 509.335,Z 263.457,A -85,B 0,C 180,E1 -5603.588,E2 -5603.588} C_VEL
LIN {X 0,Y 509.409,Z 260.79,A -85,B 0,C 180,E1 -5606.263,E2 -5606.263} C_VEL
LIN {X 0,Y 509.369,Z 258.225,A -85,B 0,C 180,E1 -5608.876,E2 -5608.876} C_VEL
LIN {X 0,Y 509.418,Z 256.659,A -85,B 0,C 180,E1 -5610.695,E2 -5610.695} C_VEL
LIN {X 0,Y 509.739,Z 256.619,A -85,B 0,C 180,E1 -5613.47,E2 -5613.47} C_VEL
LIN {X 0,Y 509.812,Z 256.604,A -85,B 0,C 180,E1 -5616.355,E2 -5616.355} C_VEL
LIN {X 0,Y 509.849,Z 256.601,A -85,B 0,C 180,E1 -5619.353,E2 -5619.353} C_VEL
LIN {X 0,Y 509.816,Z 256.604,A -85,B 0,C 180,E1 -5622.492,E2 -5622.492} C_VEL
LIN {X 0,Y 509.843,Z 256.601,A -85,B 0,C 180,E1 -5625.33,E2 -5625.33} C_VEL
LIN {X 0,Y 509.847,Z 256.602,A -85,B 0,C 180,E1 -5627.926,E2 -5627.926} C_VEL
LIN {X 0,Y 509.209,Z 256.682,A -85,B 0,C 180,E1 -5628.586,E2 -5628.586} C_VEL
LIN {X 0,Y 506.349,Z 257.039,A -85,B 0,C 180,E1 -5629.657,E2 -5629.657} C_VEL
LIN {X 0,Y 503.916,Z 257.341,A -85,B 0,C 180,E1 -5630.519,E2 -5630.519} C_VEL
LIN {X 0,Y 502.876,Z 257.47,A -85,B 0,C 180,E1 -5631.186,E2 -5631.186} C_VEL
LIN {X 0,Y 502.795,Z 257.479,A -85,B 0,C 180,E1 -5631.412,E2 -5631.412} C_VEL
LIN {X 0,Y 502.778,Z 257.483,A -85,B 0,C 180,E1 -5634.169,E2 -5634.169} C_VEL
LIN {X 0,Y 502.834,Z 257.477,A -85,B 0,C 180,E1 -5636.994,E2 -5636.994} C_VEL
LIN {X 0,Y 502.819,Z 257.48,A -85,B 0,C 180,E1 -5640.065,E2 -5640.065} C_VEL
LIN {X 0,Y 502.831,Z 257.476,A -85,B 0,C 180,E1 -5642.533,E2 -5642.533} C_VEL
LIN {X 0,Y 502.775,Z 257.481,A -85,B 0,C 180,E1 -5645.313,E2 -5645.313} C_VEL
LIN {X 0,Y 502.783,Z 257.483,A -85,B 0,C 180,E1 -5647.826,E2 -5647.826} C_VEL
LIN {X 0,Y 502.823,Z 257.479,A -85,B 0,C 180,E1 -5650.4,E2 -5650.4} C_VEL
LIN {X 0,Y 502.817,Z 257.476,A -85,B 0,C 180,E1 -5652.931,E2 -5652.931} C_VEL
LIN {X 0,Y 502.846,Z 257.475,A -85,B 0,C 180,E1 -5655.429,E2 -5655.429} C_VEL
LIN {X 0,Y 502.88,Z 257.468,A -85,B 0,C 180,E1 -5658.717,E2 -5658.717} C_VEL
LIN {X 0,Y 502.905,Z 257.466,A -85,B 0,C 180,E1 -5661.967,E2 -5661.967} C_VEL
LIN {X 0,Y 502.858,Z 257.47,A -85,B 0,C 180,E1 -5665.19,E2 -5665.19} C_VEL
LIN {X 0,Y 503.025,Z 257.453,A -85,B 0,C 180,E1 -5667.598,E2 -5667.598} C_VEL
LIN {X 0,Y 503.031,Z 257.451,A -85,B 0,C 180,E1 -5670,E2 -5670} C_VEL
LIN {X 0,Y 503.022,Z 257.451,A -85,B 0,C 180,E1 -5672.402,E2 -5672.402} C_VEL
LIN {X 0,Y 502.932,Z 257.463,A -85,B 0,C 180,E1 -5675.614,E2 -5675.614} C_VEL
LIN {X 0,Y 502.865,Z 257.469,A -85,B 0,C 180,E1 -5678.844,E2 -5678.844} C_VEL
LIN {X 0,Y 502.85,Z 257.474,A -85,B 0,C 180,E1 -5682.102,E2 -5682.102} C_VEL
LIN {X 0,Y 502.852,Z 257.474,A -85,B 0,C 180,E1 -5685.4,E2 -5685.4} C_VEL
LIN {X 0,Y 502.83,Z 257.477,A -85,B 0,C 180,E1 -5688.752,E2 -5688.752} C_VEL
LIN {X 0,Y 502.787,Z 257.481,A -85,B 0,C 180,E1 -5691.311,E2 -5691.311} C_VEL
LIN {X 0,Y 502.787,Z 257.48,A -85,B 0,C 180,E1 -5693.914,E2 -5693.914} C_VEL
LIN {X 0,Y 502.868,Z 257.472,A -85,B 0,C 180,E1 -5696.566,E2 -5696.566} C_VEL
LIN {X 0,Y 502.825,Z 257.48,A -85,B 0,C 180,E1 -5699.288,E2 -5699.288} C_VEL
LIN {X 0,Y 502.787,Z 257.483,A -85,B 0,C 180,E1 -5702.085,E2 -5702.085} C_VEL
LIN {X 0,Y 502.8,Z 257.479,A -85,B 0,C 180,E1 -5704.966,E2 -5704.966} C_VEL
LIN {X 0,Y 502.797,Z 257.482,A -85,B 0,C 180,E1 -5708.486,E2 -5708.486} C_VEL
LIN {X 0,Y 502.77,Z 257.484,A -85,B 0,C 180,E1 -5711.071,E2 -5711.071} C_VEL
LIN {X 0,Y 502.789,Z 257.483,A -85,B 0,C 180,E1 -5714.53,E2 -5714.53} C_VEL
LIN {X 0,Y 502.799,Z 257.48,A -85,B 0,C 180,E1 -5717.861,E2 -5717.861} C_VEL
LIN {X 0,Y 502.805,Z 257.479,A -85,B 0,C 180,E1 -5721.024,E2 -5721.024} C_VEL
LIN {X 0,Y 502.779,Z 257.482,A -85,B 0,C 180,E1 -5724.169,E2 -5724.169} C_VEL
LIN {X 0,Y 502.835,Z 257.476,A -85,B 0,C 180,E1 -5726.994,E2 -5726.994} C_VEL
LIN {X 0,Y 502.82,Z 257.479,A -85,B 0,C 180,E1 -5730.065,E2 -5730.065} C_VEL
LIN {X 0,Y 502.832,Z 257.477,A -85,B 0,C 180,E1 -5732.533,E2 -5732.533} C_VEL
LIN {X 0,Y 502.789,Z 257.48,A -85,B 0,C 180,E1 -5735.31,E2 -5735.31} C_VEL
LIN {X 0,Y 502.785,Z 257.482,A -85,B 0,C 180,E1 -5737.826,E2 -5737.826} C_VEL
LIN {X 0,Y 502.824,Z 257.48,A -85,B 0,C 180,E1 -5740.4,E2 -5740.4} C_VEL
LIN {X 0,Y 502.818,Z 257.477,A -85,B 0,C 180,E1 -5742.931,E2 -5742.931} C_VEL
LIN {X 0,Y 502.843,Z 257.474,A -85,B 0,C 180,E1 -5745.429,E2 -5745.429} C_VEL
LIN {X 0,Y 502.883,Z 257.468,A -85,B 0,C 180,E1 -5748.717,E2 -5748.717} C_VEL
LIN {X 0,Y 502.877,Z 257.469,A -85,B 0,C 180,E1 -5751.966,E2 -5751.966} C_VEL
LIN {X 0,Y 502.902,Z 257.467,A -85,B 0,C 180,E1 -5754.386,E2 -5754.386} C_VEL
LIN {X 0,Y 503.026,Z 257.452,A -85,B 0,C 180,E1 -5757.598,E2 -5757.598} C_VEL
LIN {X 0,Y 503.032,Z 257.452,A -85,B 0,C 180,E1 -5760,E2 -5760} C_VEL
LIN {X 0,Y 503.028,Z 257.45,A -85,B 0,C 180,E1 -5762.402,E2 -5762.402} C_VEL
LIN {X 0,Y 502.93,Z 257.463,A -85,B 0,C 180,E1 -5765.613,E2 -5765.613} C_VEL
LIN {X 0,Y 502.855,Z 257.471,A -85,B 0,C 180,E1 -5768.843,E2 -5768.843} C_VEL
LIN {X 0,Y 502.85,Z 257.475,A -85,B 0,C 180,E1 -5772.101,E2 -5772.101} C_VEL
LIN {X 0,Y 502.853,Z 257.475,A -85,B 0,C 180,E1 -5775.399,E2 -5775.399} C_VEL
LIN {X 0,Y 502.831,Z 257.477,A -85,B 0,C 180,E1 -5778.752,E2 -5778.752} C_VEL
LIN {X 0,Y 502.785,Z 257.482,A -85,B 0,C 180,E1 -5781.311,E2 -5781.311} C_VEL
LIN {X 0,Y 502.777,Z 257.482,A -85,B 0,C 180,E1 -5783.914,E2 -5783.914} C_VEL
LIN {X 0,Y 502.837,Z 257.475,A -85,B 0,C 180,E1 -5786.567,E2 -5786.567} C_VEL
LIN {X 0,Y 502.813,Z 257.477,A -85,B 0,C 180,E1 -5789.934,E2 -5789.934} C_VEL
LIN {X 0,Y 502.833,Z 257.475,A -85,B 0,C 180,E1 -5793.031,E2 -5793.031} C_VEL
LIN {X 0,Y 502.774,Z 257.482,A -85,B 0,C 180,E1 -5795.951,E2 -5795.951} C_VEL
LIN {X 0,Y 502.803,Z 257.476,A -85,B 0,C 180,E1 -5798.976,E2 -5798.976} C_VEL
LIN {X 0,Y 502.772,Z 257.485,A -85,B 0,C 180,E1 -5802.195,E2 -5802.195} C_VEL
LIN {X 0,Y 502.771,Z 257.517,A -85,B 0,C 180,E1 -5802.957,E2 -5802.957} C_VEL
LIN {X 0,Y 503.845,Z 263.068,A -85,B 0,C 180,E1 -5805.778,E2 -5805.778} C_VEL
LIN {X 0,Y 504.584,Z 267.821,A -85,B 0,C 180,E1 -5808.044,E2 -5808.044} C_VEL
LIN {X 0,Y 504.557,Z 272.632,A -85,B 0,C 180,E1 -5810.153,E2 -5810.153} C_VEL
LIN {X 0,Y 504.247,Z 279.896,A -85,B 0,C 180,E1 -5813.179,E2 -5813.179} C_VEL
LIN {X 0,Y 503.916,Z 287.294,A -85,B 0,C 180,E1 -5816.091,E2 -5816.091} C_VEL
LIN {X 0,Y 503.61,Z 296.037,A -85,B 0,C 180,E1 -5819.378,E2 -5819.378} C_VEL
LIN {X 0,Y 503.365,Z 303.514,A -85,B 0,C 180,E1 -5822.113,E2 -5822.113} C_VEL
LIN {X 0,Y 503.133,Z 311.056,A -85,B 0,C 180,E1 -5824.783,E2 -5824.783} C_VEL
LIN {X 0,Y 502.892,Z 319.72,A -85,B 0,C 180,E1 -5827.831,E2 -5827.831} C_VEL
LIN {X 0,Y 502.728,Z 325.421,A -85,B 0,C 180,E1 -5829.802,E2 -5829.802} C_VEL
LIN {X 0,Y 506.991,Z 342.639,A -85,B 0,C 180,E1 -5830.312,E2 -5830.312} C_VEL
LIN {X 0,Y 507.277,Z 346.649,A -85,B 0,C 180,E1 -5830.432,E2 -5830.432} C_VEL
LIN {X 0,Y 506.879,Z 361.359,A -85,B 0,C 180,E1 -5830.91,E2 -5830.91} C_VEL
LIN {X 0,Y 506.262,Z 376.82,A -85,B 0,C 180,E1 -5831.59,E2 -5831.59} C_VEL
LIN {X 0,Y 505.692,Z 391.108,A -85,B 0,C 180,E1 -5832.405,E2 -5832.405} C_VEL
LIN {X 0,Y 505.117,Z 404.099,A -85,B 0,C 180,E1 -5833.323,E2 -5833.323} C_VEL
LIN {X 0,Y 504.524,Z 415.954,A -85,B 0,C 180,E1 -5834.331,E2 -5834.331} C_VEL
LIN {X 0,Y 503.967,Z 427.153,A -85,B 0,C 180,E1 -5835.462,E2 -5835.462} C_VEL
LIN {X 0,Y 503.472,Z 437.361,A -85,B 0,C 180,E1 -5836.684,E2 -5836.684} C_VEL
LIN {X 0,Y 502.966,Z 447.608,A -85,B 0,C 180,E1 -5838.149,E2 -5838.149} C_VEL
LIN {X 0,Y 502.737,Z 455.64,A -85,B 0,C 180,E1 -5839.529,E2 -5839.529} C_VEL
LIN {X 0,Y 502.436,Z 463.41,A -85,B 0,C 180,E1 -5841.149,E2 -5841.149} C_VEL
LIN {X 0,Y 502.244,Z 469.6,A -85,B 0,C 180,E1 -5842.765,E2 -5842.765} C_VEL
LIN {X 0,Y 502.199,Z 474.388,A -85,B 0,C 180,E1 -5844.378,E2 -5844.378} C_VEL
LIN {X 0,Y 502.096,Z 477.894,A -85,B 0,C 180,E1 -5845.987,E2 -5845.987} C_VEL
LIN {X 0,Y 502.062,Z 480.196,A -85,B 0,C 180,E1 -5847.593,E2 -5847.593} C_VEL
LIN {X 0,Y 501.987,Z 481.352,A -85,B 0,C 180,E1 -5849.198,E2 -5849.198} C_VEL
LIN {X 0,Y 501.987,Z 481.35,A -85,B 0,C 180,E1 -5850.802,E2 -5850.802} C_VEL
LIN {X 0,Y 502.062,Z 480.191,A -85,B 0,C 180,E1 -5852.407,E2 -5852.407} C_VEL
LIN {X 0,Y 502.096,Z 477.889,A -85,B 0,C 180,E1 -5854.013,E2 -5854.013} C_VEL
LIN {X 0,Y 502.201,Z 474.387,A -85,B 0,C 180,E1 -5855.622,E2 -5855.622} C_VEL
LIN {X 0,Y 502.245,Z 469.602,A -85,B 0,C 180,E1 -5857.235,E2 -5857.235} C_VEL
LIN {X 0,Y 502.436,Z 463.407,A -85,B 0,C 180,E1 -5858.851,E2 -5858.851} C_VEL
LIN {X 0,Y 502.737,Z 455.634,A -85,B 0,C 180,E1 -5860.471,E2 -5860.471} C_VEL
LIN {X 0,Y 503.016,Z 446.43,A -85,B 0,C 180,E1 -5862.035,E2 -5862.035} C_VEL
LIN {X 0,Y 503.472,Z 437.358,A -85,B 0,C 180,E1 -5863.316,E2 -5863.316} C_VEL
LIN {X 0,Y 503.951,Z 427.156,A -85,B 0,C 180,E1 -5864.538,E2 -5864.538} C_VEL
LIN {X 0,Y 504.51,Z 416.075,A -85,B 0,C 180,E1 -5865.66,E2 -5865.66} C_VEL
LIN {X 0,Y 505.08,Z 404.12,A -85,B 0,C 180,E1 -5866.678,E2 -5866.678} C_VEL
LIN {X 0,Y 505.658,Z 391.126,A -85,B 0,C 180,E1 -5867.596,E2 -5867.596} C_VEL
LIN {X 0,Y 506.268,Z 376.836,A -85,B 0,C 180,E1 -5868.41,E2 -5868.41} C_VEL
LIN {X 0,Y 506.858,Z 361.372,A -85,B 0,C 180,E1 -5869.091,E2 -5869.091} C_VEL
LIN {X 0,Y 507.258,Z 345.98,A -85,B 0,C 180,E1 -5869.588,E2 -5869.588} C_VEL
LIN {X 0,Y 507.08,Z 342.936,A -85,B 0,C 180,E1 -5869.679,E2 -5869.679} C_VEL
LIN {X 0,Y 502.895,Z 326.465,A -85,B 0,C 180,E1 -5870.172,E2 -5870.172} C_VEL
LIN {X 0,Y 502.73,Z 325.365,A -85,B 0,C 180,E1 -5870.217,E2 -5870.217} C_VEL
LIN {X 0,Y 502.967,Z 317.245,A -85,B 0,C 180,E1 -5873.032,E2 -5873.032} C_VEL
LIN {X 0,Y 503.23,Z 308.58,A -85,B 0,C 180,E1 -5876.099,E2 -5876.099} C_VEL
LIN {X 0,Y 503.446,Z 299.313,A -85,B 0,C 180,E1 -5879.248,E2 -5879.248} C_VEL
LIN {X 0,Y 503.589,Z 291.369,A -85,B 0,C 180,E1 -5882.027,E2 -5882.027} C_VEL
LIN {X 0,Y 503.853,Z 283.647,A -85,B 0,C 180,E1 -5884.882,E2 -5884.882} C_VEL
LIN {X 0,Y 504.159,Z 276.552,A -85,B 0,C 180,E1 -5887.833,E2 -5887.833} C_VEL
LIN {X 0,Y 504.468,Z 272.102,A -85,B 0,C 180,E1 -5889.983,E2 -5889.983} C_VEL
LIN {X 0,Y 504.624,Z 268.738,A -85,B 0,C 180,E1 -5891.952,E2 -5891.952} C_VEL
LIN {X 0,Y 504.318,Z 266.021,A -85,B 0,C 180,E1 -5894.17,E2 -5894.17} C_VEL
LIN {X 0,Y 503.97,Z 264.398,A -85,B 0,C 180,E1 -5896.482,E2 -5896.482} C_VEL
LIN {X 0,Y 503.765,Z 263.979,A -85,B 0,C 180,E1 -5897.96,E2 -5897.96} C_VEL
LIN {X 0,Y 503.265,Z 264.328,A -85,B 0,C 180,E1 -5901.067,E2 -5901.067} C_VEL
LIN {X 0,Y 503,Z 265.574,A -85,B 0,C 180,E1 -5904.068,E2 -5904.068} C_VEL
LIN {X 0,Y 502.795,Z 267.256,A -85,B 0,C 180,E1 -5907.001,E2 -5907.001} C_VEL
LIN {X 0,Y 502.662,Z 269.307,A -85,B 0,C 180,E1 -5910.096,E2 -5910.096} C_VEL
LIN {X 0,Y 502.541,Z 271.055,A -85,B 0,C 180,E1 -5912.516,E2 -5912.516} C_VEL
LIN {X 0,Y 502.439,Z 273.274,A -85,B 0,C 180,E1 -5915.397,E2 -5915.397} C_VEL
LIN {X 0,Y 502.42,Z 273.884,A -85,B 0,C 180,E1 -5916.157,E2 -5916.157} C_VEL
LIN {X 0,Y 506.635,Z 288.57,A -85,B 0,C 180,E1 -5916.657,E2 -5916.657} C_VEL
LIN {X 0,Y 506.439,Z 303.222,A -85,B 0,C 180,E1 -5917.135,E2 -5917.135} C_VEL
LIN {X 0,Y 505.996,Z 318.703,A -85,B 0,C 180,E1 -5917.814,E2 -5917.814} C_VEL
LIN {X 0,Y 505.472,Z 332.978,A -85,B 0,C 180,E1 -5918.616,E2 -5918.616} C_VEL
LIN {X 0,Y 504.978,Z 346.164,A -85,B 0,C 180,E1 -5919.533,E2 -5919.533} C_VEL
LIN {X 0,Y 504.439,Z 358.499,A -85,B 0,C 180,E1 -5920.571,E2 -5920.571} C_VEL
LIN {X 0,Y 504,Z 368.973,A -85,B 0,C 180,E1 -5921.621,E2 -5921.621} C_VEL
LIN {X 0,Y 503.486,Z 380.128,A -85,B 0,C 180,E1 -5922.955,E2 -5922.955} C_VEL
LIN {X 0,Y 503.123,Z 389.053,A -85,B 0,C 180,E1 -5924.235,E2 -5924.235} C_VEL
LIN {X 0,Y 502.793,Z 397.217,A -85,B 0,C 180,E1 -5925.635,E2 -5925.635} C_VEL
LIN {X 0,Y 502.519,Z 404.159,A -85,B 0,C 180,E1 -5927.07,E2 -5927.07} C_VEL
LIN {X 0,Y 502.315,Z 410.523,A -85,B 0,C 180,E1 -5928.704,E2 -5928.704} C_VEL
LIN {X 0,Y 502.155,Z 415.421,A -85,B 0,C 180,E1 -5930.332,E2 -5930.332} C_VEL
LIN {X 0,Y 502.124,Z 418.969,A -85,B 0,C 180,E1 -5931.954,E2 -5931.954} C_VEL
LIN {X 0,Y 502.169,Z 421.315,A -85,B 0,C 180,E1 -5933.572,E2 -5933.572} C_VEL
LIN {X 0,Y 502.052,Z 422.465,A -85,B 0,C 180,E1 -5935.182,E2 -5935.182} C_VEL
LIN {X 0,Y 502.1,Z 422.465,A -85,B 0,C 180,E1 -5936.791,E2 -5936.791} C_VEL
LIN {X 0,Y 502.035,Z 421.376,A -85,B 0,C 180,E1 -5938.396,E2 -5938.396} C_VEL
LIN {X 0,Y 502.002,Z 419.101,A -85,B 0,C 180,E1 -5940,E2 -5940} C_VEL
LIN {X 0,Y 502.083,Z 415.655,A -85,B 0,C 180,E1 -5941.604,E2 -5941.604} C_VEL
LIN {X 0,Y 502.33,Z 410.933,A -85,B 0,C 180,E1 -5943.208,E2 -5943.208} C_VEL
LIN {X 0,Y 502.528,Z 404.795,A -85,B 0,C 180,E1 -5944.814,E2 -5944.814} C_VEL
LIN {X 0,Y 502.703,Z 397.153,A -85,B 0,C 180,E1 -5946.422,E2 -5946.422} C_VEL
LIN {X 0,Y 503.092,Z 388.924,A -85,B 0,C 180,E1 -5947.828,E2 -5947.828} C_VEL
LIN {X 0,Y 503.522,Z 379.072,A -85,B 0,C 180,E1 -5949.237,E2 -5949.237} C_VEL
LIN {X 0,Y 503.991,Z 368.989,A -85,B 0,C 180,E1 -5950.445,E2 -5950.445} C_VEL
LIN {X 0,Y 504.556,Z 356.942,A -85,B 0,C 180,E1 -5951.653,E2 -5951.653} C_VEL
LIN {X 0,Y 505.197,Z 343.626,A -85,B 0,C 180,E1 -5952.759,E2 -5952.759} C_VEL
LIN {X 0,Y 505.633,Z 331.68,A -85,B 0,C 180,E1 -5953.58,E2 -5953.58} C_VEL
LIN {X 0,Y 506.16,Z 317.6,A -85,B 0,C 180,E1 -5954.371,E2 -5954.371} C_VEL
LIN {X 0,Y 506.64,Z 302.825,A -85,B 0,C 180,E1 -5955.02,E2 -5955.02} C_VEL
LIN {X 0,Y 506.788,Z 288.296,A -85,B 0,C 180,E1 -5955.504,E2 -5955.504} C_VEL
LIN {X 0,Y 503.151,Z 275.21,A -85,B 0,C 180,E1 -5955.954,E2 -5955.954} C_VEL
LIN {X 0,Y 502.202,Z 271.627,A -85,B 0,C 180,E1 -5956.076,E2 -5956.076} C_VEL
LIN {X 0,Y 502.198,Z 268.859,A -85,B 0,C 180,E1 -5958.776,E2 -5958.776} C_VEL
LIN {X 0,Y 502.206,Z 266.304,A -85,B 0,C 180,E1 -5961.337,E2 -5961.337} C_VEL
LIN {X 0,Y 502.267,Z 263.724,A -85,B 0,C 180,E1 -5963.941,E2 -5963.941} C_VEL
LIN {X 0,Y 502.337,Z 261.122,A -85,B 0,C 180,E1 -5966.596,E2 -5966.596} C_VEL
LIN {X 0,Y 502.343,Z 257.941,A -85,B 0,C 180,E1 -5969.841,E2 -5969.841} C_VEL
LIN {X 0,Y 502.344,Z 257.554,A -85,B 0,C 180,E1 -5970.242,E2 -5970.242} C_VEL
LIN {X 0,Y 502.652,Z 257.502,A -85,B 0,C 180,E1 -5973.045,E2 -5973.045} C_VEL
LIN {X 0,Y 502.784,Z 257.481,A -85,B 0,C 180,E1 -5974.967,E2 -5974.967} C_VEL
LIN {X 0,Y 502.798,Z 257.481,A -85,B 0,C 180,E1 -5978.486,E2 -5978.486} C_VEL
LIN {X 0,Y 502.803,Z 257.479,A -85,B 0,C 180,E1 -5981.068,E2 -5981.068} C_VEL
LIN {X 0,Y 502.782,Z 257.481,A -85,B 0,C 180,E1 -5984.34,E2 -5984.34} C_VEL
LIN {X 0,Y 502.776,Z 257.482,A -85,B 0,C 180,E1 -5986.769,E2 -5986.769} C_VEL
LIN {X 0,Y 502.822,Z 257.478,A -85,B 0,C 180,E1 -5989.005,E2 -5989.005} C_VEL
LIN {X 0,Y 502.795,Z 257.479,A -85,B 0,C 180,E1 -5991.412,E2 -5991.412} C_VEL
LIN {X 0,Y 502.134,Z 257.564,A -85,B 0,C 180,E1 -5992.08,E2 -5992.08} C_VEL
LIN {X 0,Y 499.268,Z 257.919,A -85,B 0,C 180,E1 -5993.166,E2 -5993.166} C_VEL
LIN {X 0,Y 496.848,Z 258.223,A -85,B 0,C 180,E1 -5994.04,E2 -5994.04} C_VEL
LIN {X 0,Y 495.822,Z 258.348,A -85,B 0,C 180,E1 -5994.716,E2 -5994.716} C_VEL
LIN {X 0,Y 495.746,Z 258.357,A -85,B 0,C 180,E1 -5994.945,E2 -5994.945} C_VEL
LIN {X 0,Y 495.769,Z 258.353,A -85,B 0,C 180,E1 -5997.406,E2 -5997.406} C_VEL
LIN {X 0,Y 495.77,Z 258.357,A -85,B 0,C 180,E1 -6000.254,E2 -6000.254} C_VEL
LIN {X 0,Y 495.809,Z 258.35,A -85,B 0,C 180,E1 -6003.255,E2 -6003.255} C_VEL
LIN {X 0,Y 495.743,Z 258.358,A -85,B 0,C 180,E1 -6006.612,E2 -6006.612} C_VEL
LIN {X 0,Y 495.782,Z 258.354,A -85,B 0,C 180,E1 -6009.324,E2 -6009.324} C_VEL
LIN {X 0,Y 495.782,Z 258.353,A -85,B 0,C 180,E1 -6011.828,E2 -6011.828} C_VEL
LIN {X 0,Y 495.827,Z 258.348,A -85,B 0,C 180,E1 -6014.548,E2 -6014.548} C_VEL
LIN {X 0,Y 495.832,Z 258.348,A -85,B 0,C 180,E1 -6017.965,E2 -6017.965} C_VEL
LIN {X 0,Y 495.842,Z 258.348,A -85,B 0,C 180,E1 -6021.03,E2 -6021.03} C_VEL
LIN {X 0,Y 495.861,Z 258.346,A -85,B 0,C 180,E1 -6024.306,E2 -6024.306} C_VEL
LIN {X 0,Y 495.992,Z 258.33,A -85,B 0,C 180,E1 -6027.564,E2 -6027.564} C_VEL
LIN {X 0,Y 496.002,Z 258.327,A -85,B 0,C 180,E1 -6030,E2 -6030} C_VEL
LIN {X 0,Y 495.99,Z 258.327,A -85,B 0,C 180,E1 -6032.436,E2 -6032.436} C_VEL
LIN {X 0,Y 495.887,Z 258.34,A -85,B 0,C 180,E1 -6035.694,E2 -6035.694} C_VEL
LIN {X 0,Y 495.835,Z 258.345,A -85,B 0,C 180,E1 -6038.97,E2 -6038.97} C_VEL
LIN {X 0,Y 495.832,Z 258.348,A -85,B 0,C 180,E1 -6042.035,E2 -6042.035} C_VEL
LIN {X 0,Y 495.827,Z 258.35,A -85,B 0,C 180,E1 -6045.451,E2 -6045.451} C_VEL
LIN {X 0,Y 495.786,Z 258.354,A -85,B 0,C 180,E1 -6049.029,E2 -6049.029} C_VEL
LIN {X 0,Y 495.746,Z 258.362,A -85,B 0,C 180,E1 -6051.629,E2 -6051.629} C_VEL
LIN {X 0,Y 495.782,Z 258.356,A -85,B 0,C 180,E1 -6054.873,E2 -6054.873} C_VEL
LIN {X 0,Y 495.815,Z 258.349,A -85,B 0,C 180,E1 -6056.974,E2 -6056.974} C_VEL
LIN {X 0,Y 495.766,Z 258.354,A -85,B 0,C 180,E1 -6060.147,E2 -6060.147} C_VEL
LIN {X 0,Y 495.797,Z 258.352,A -85,B 0,C 180,E1 -6063.244,E2 -6063.244} C_VEL
LIN {X 0,Y 495.715,Z 258.359,A -85,B 0,C 180,E1 -6066.087,E2 -6066.087} C_VEL
LIN {X 0,Y 495.764,Z 258.357,A -85,B 0,C 180,E1 -6068.768,E2 -6068.768} C_VEL
LIN {X 0,Y 495.727,Z 258.36,A -85,B 0,C 180,E1 -6071.785,E2 -6071.785} C_VEL
LIN {X 0,Y 495.741,Z 258.358,A -85,B 0,C 180,E1 -6075.141,E2 -6075.141} C_VEL
LIN {X 0,Y 495.76,Z 258.355,A -85,B 0,C 180,E1 -6078.219,E2 -6078.219} C_VEL
LIN {X 0,Y 495.753,Z 258.356,A -85,B 0,C 180,E1 -6081.408,E2 -6081.408} C_VEL
LIN {X 0,Y 495.751,Z 258.357,A -85,B 0,C 180,E1 -6084.462,E2 -6084.462} C_VEL
LIN {X 0,Y 495.771,Z 258.353,A -85,B 0,C 180,E1 -6087.406,E2 -6087.406} C_VEL
LIN {X 0,Y 495.771,Z 258.355,A -85,B 0,C 180,E1 -6090.254,E2 -6090.254} C_VEL
LIN {X 0,Y 495.811,Z 258.348,A -85,B 0,C 180,E1 -6093.255,E2 -6093.255} C_VEL
LIN {X 0,Y 495.748,Z 258.358,A -85,B 0,C 180,E1 -6096.612,E2 -6096.612} C_VEL
LIN {X 0,Y 495.784,Z 258.353,A -85,B 0,C 180,E1 -6099.324,E2 -6099.324} C_VEL
LIN {X 0,Y 495.784,Z 258.354,A -85,B 0,C 180,E1 -6101.828,E2 -6101.828} C_VEL
LIN {X 0,Y 495.829,Z 258.348,A -85,B 0,C 180,E1 -6104.548,E2 -6104.548} C_VEL
LIN {X 0,Y 495.834,Z 258.349,A -85,B 0,C 180,E1 -6107.965,E2 -6107.965} C_VEL
LIN {X 0,Y 495.84,Z 258.348,A -85,B 0,C 180,E1 -6111.03,E2 -6111.03} C_VEL
LIN {X 0,Y 495.86,Z 258.345,A -85,B 0,C 180,E1 -6114.306,E2 -6114.306} C_VEL
LIN {X 0,Y 495.993,Z 258.328,A -85,B 0,C 180,E1 -6117.563,E2 -6117.563} C_VEL
LIN {X 0,Y 496.003,Z 258.328,A -85,B 0,C 180,E1 -6120,E2 -6120} C_VEL
LIN {X 0,Y 495.997,Z 258.326,A -85,B 0,C 180,E1 -6122.436,E2 -6122.436} C_VEL
LIN {X 0,Y 495.885,Z 258.34,A -85,B 0,C 180,E1 -6125.693,E2 -6125.693} C_VEL
LIN {X 0,Y 495.813,Z 258.349,A -85,B 0,C 180,E1 -6128.97,E2 -6128.97} C_VEL
LIN {X 0,Y 495.833,Z 258.348,A -85,B 0,C 180,E1 -6132.034,E2 -6132.034} C_VEL
LIN {X 0,Y 495.828,Z 258.351,A -85,B 0,C 180,E1 -6135.451,E2 -6135.451} C_VEL
LIN {X 0,Y 495.783,Z 258.356,A -85,B 0,C 180,E1 -6138.237,E2 -6138.237} C_VEL
LIN {X 0,Y 495.778,Z 258.352,A -85,B 0,C 180,E1 -6140.756,E2 -6140.756} C_VEL
LIN {X 0,Y 495.745,Z 258.359,A -85,B 0,C 180,E1 -6143.387,E2 -6143.387} C_VEL
LIN {X 0,Y 495.752,Z 258.361,A -85,B 0,C 180,E1 -6146.07,E2 -6146.07} C_VEL
LIN {X 0,Y 495.731,Z 258.359,A -85,B 0,C 180,E1 -6148.817,E2 -6148.817} C_VEL
LIN {X 0,Y 495.757,Z 258.357,A -85,B 0,C 180,E1 -6151.725,E2 -6151.725} C_VEL
LIN {X 0,Y 495.767,Z 258.355,A -85,B 0,C 180,E1 -6154.693,E2 -6154.693} C_VEL
LIN {X 0,Y 495.731,Z 258.358,A -85,B 0,C 180,E1 -6157.561,E2 -6157.561} C_VEL
LIN {X 0,Y 495.756,Z 258.357,A -85,B 0,C 180,E1 -6160.046,E2 -6160.046} C_VEL
LIN {X 0,Y 495.741,Z 258.429,A -85,B 0,C 180,E1 -6162.548,E2 -6162.548} C_VEL
LIN {X 0,Y 496.873,Z 264.307,A -85,B 0,C 180,E1 -6165.585,E2 -6165.585} C_VEL
LIN {X 0,Y 497.624,Z 269.01,A -85,B 0,C 180,E1 -6167.867,E2 -6167.867} C_VEL
LIN {X 0,Y 497.66,Z 273.072,A -85,B 0,C 180,E1 -6169.693,E2 -6169.693} C_VEL
LIN {X 0,Y 497.291,Z 281.069,A -85,B 0,C 180,E1 -6173.084,E2 -6173.084} C_VEL
LIN {X 0,Y 496.928,Z 288.44,A -85,B 0,C 180,E1 -6176.038,E2 -6176.038} C_VEL
LIN {X 0,Y 496.598,Z 297.152,A -85,B 0,C 180,E1 -6179.37,E2 -6179.37} C_VEL
LIN {X 0,Y 496.344,Z 304.607,A -85,B 0,C 180,E1 -6182.143,E2 -6182.143} C_VEL
LIN {X 0,Y 496.085,Z 312.851,A -85,B 0,C 180,E1 -6185.051,E2 -6185.051} C_VEL
LIN {X 0,Y 495.826,Z 322.196,A -85,B 0,C 180,E1 -6188.375,E2 -6188.375} C_VEL
LIN {X 0,Y 495.719,Z 325.424,A -85,B 0,C 180,E1 -6189.505,E2 -6189.505} C_VEL
LIN {X 0,Y 499.878,Z 342.02,A -85,B 0,C 180,E1 -6190.006,E2 -6190.006} C_VEL
LIN {X 0,Y 500.596,Z 346.548,A -85,B 0,C 180,E1 -6190.157,E2 -6190.157} C_VEL
LIN {X 0,Y 500.154,Z 360.724,A -85,B 0,C 180,E1 -6190.617,E2 -6190.617} C_VEL
LIN {X 0,Y 499.585,Z 375.805,A -85,B 0,C 180,E1 -6191.281,E2 -6191.281} C_VEL
LIN {X 0,Y 498.955,Z 389.488,A -85,B 0,C 180,E1 -6192.054,E2 -6192.054} C_VEL
LIN {X 0,Y 498.309,Z 402.77,A -85,B 0,C 180,E1 -6192.983,E2 -6192.983} C_VEL
LIN {X 0,Y 497.669,Z 415.17,A -85,B 0,C 180,E1 -6194.035,E2 -6194.035} C_VEL
LIN {X 0,Y 497.044,Z 427.15,A -85,B 0,C 180,E1 -6195.255,E2 -6195.255} C_VEL
LIN {X 0,Y 496.521,Z 437.358,A -85,B 0,C 180,E1 -6196.494,E2 -6196.494} C_VEL
LIN {X 0,Y 495.986,Z 446.987,A -85,B 0,C 180,E1 -6197.88,E2 -6197.88} C_VEL
LIN {X 0,Y 495.71,Z 455.638,A -85,B 0,C 180,E1 -6199.379,E2 -6199.379} C_VEL
LIN {X 0,Y 495.358,Z 463.408,A -85,B 0,C 180,E1 -6201.021,E2 -6201.021} C_VEL
LIN {X 0,Y 495.168,Z 469.599,A -85,B 0,C 180,E1 -6202.661,E2 -6202.661} C_VEL
LIN {X 0,Y 495.115,Z 474.387,A -85,B 0,C 180,E1 -6204.297,E2 -6204.297} C_VEL
LIN {X 0,Y 494.993,Z 477.894,A -85,B 0,C 180,E1 -6205.929,E2 -6205.929} C_VEL
LIN {X 0,Y 494.97,Z 480.197,A -85,B 0,C 180,E1 -6207.559,E2 -6207.559} C_VEL
LIN {X 0,Y 494.907,Z 481.352,A -85,B 0,C 180,E1 -6209.186,E2 -6209.186} C_VEL
LIN {X 0,Y 494.907,Z 481.35,A -85,B 0,C 180,E1 -6210.814,E2 -6210.814} C_VEL
LIN {X 0,Y 494.97,Z 480.191,A -85,B 0,C 180,E1 -6212.441,E2 -6212.441} C_VEL
LIN {X 0,Y 494.993,Z 477.888,A -85,B 0,C 180,E1 -6214.071,E2 -6214.071} C_VEL
LIN {X 0,Y 495.118,Z 474.386,A -85,B 0,C 180,E1 -6215.702,E2 -6215.702} C_VEL
LIN {X 0,Y 495.169,Z 469.601,A -85,B 0,C 180,E1 -6217.339,E2 -6217.339} C_VEL
LIN {X 0,Y 495.358,Z 463.406,A -85,B 0,C 180,E1 -6218.979,E2 -6218.979} C_VEL
LIN {X 0,Y 495.709,Z 455.632,A -85,B 0,C 180,E1 -6220.621,E2 -6220.621} C_VEL
LIN {X 0,Y 495.992,Z 446.965,A -85,B 0,C 180,E1 -6222.123,E2 -6222.123} C_VEL
LIN {X 0,Y 496.521,Z 437.356,A -85,B 0,C 180,E1 -6223.506,E2 -6223.506} C_VEL
LIN {X 0,Y 497.009,Z 427.153,A -85,B 0,C 180,E1 -6224.746,E2 -6224.746} C_VEL
LIN {X 0,Y 497.656,Z 415.319,A -85,B 0,C 180,E1 -6225.952,E2 -6225.952} C_VEL
LIN {X 0,Y 498.315,Z 402.774,A -85,B 0,C 180,E1 -6227.017,E2 -6227.017} C_VEL
LIN {X 0,Y 498.984,Z 389.48,A -85,B 0,C 180,E1 -6227.945,E2 -6227.945} C_VEL
LIN {X 0,Y 499.586,Z 375.803,A -85,B 0,C 180,E1 -6228.719,E2 -6228.719} C_VEL
LIN {X 0,Y 500.132,Z 361.864,A -85,B 0,C 180,E1 -6229.339,E2 -6229.339} C_VEL
LIN {X 0,Y 500.545,Z 347.22,A -85,B 0,C 180,E1 -6229.826,E2 -6229.826} C_VEL
LIN {X 0,Y 500.402,Z 344.363,A -85,B 0,C 180,E1 -6229.913,E2 -6229.913} C_VEL
LIN {X 0,Y 496.449,Z 328.501,A -85,B 0,C 180,E1 -6230.415,E2 -6230.415} C_VEL
LIN {X 0,Y 495.719,Z 325.386,A -85,B 0,C 180,E1 -6230.509,E2 -6230.509} C_VEL
LIN {X 0,Y 495.947,Z 317.245,A -85,B 0,C 180,E1 -6233.377,E2 -6233.377} C_VEL
LIN {X 0,Y 496.189,Z 309.602,A -85,B 0,C 180,E1 -6236.046,E2 -6236.046} C_VEL
LIN {X 0,Y 496.401,Z 300.184,A -85,B 0,C 180,E1 -6239.239,E2 -6239.239} C_VEL
LIN {X 0,Y 496.547,Z 292.779,A -85,B 0,C 180,E1 -6241.873,E2 -6241.873} C_VEL
LIN {X 0,Y 496.833,Z 284.843,A -85,B 0,C 180,E1 -6244.871,E2 -6244.871} C_VEL
LIN {X 0,Y 497.151,Z 278.261,A -85,B 0,C 180,E1 -6247.661,E2 -6247.661} C_VEL
LIN {X 0,Y 497.544,Z 272.967,A -85,B 0,C 180,E1 -6250.291,E2 -6250.291} C_VEL
LIN {X 0,Y 497.676,Z 270.797,A -85,B 0,C 180,E1 -6251.584,E2 -6251.584} C_VEL
LIN {X 0,Y 497.62,Z 269.157,A -85,B 0,C 180,E1 -6252.743,E2 -6252.743} C_VEL
LIN {X 0,Y 497.234,Z 266.81,A -85,B 0,C 180,E1 -6255.032,E2 -6255.032} C_VEL
LIN {X 0,Y 496.897,Z 265.582,A -85,B 0,C 180,E1 -6257.348,E2 -6257.348} C_VEL
LIN {X 0,Y 496.446,Z 265.419,A -85,B 0,C 180,E1 -6259.859,E2 -6259.859} C_VEL
LIN {X 0,Y 496.154,Z 266.084,A -85,B 0,C 180,E1 -6262.49,E2 -6262.49} C_VEL
LIN {X 0,Y 495.868,Z 267.487,A -85,B 0,C 180,E1 -6265.464,E2 -6265.464} C_VEL
LIN {X 0,Y 495.708,Z 269.197,A -85,B 0,C 180,E1 -6268.361,E2 -6268.361} C_VEL
LIN {X 0,Y 495.566,Z 271.35,A -85,B 0,C 180,E1 -6271.555,E2 -6271.555} C_VEL
LIN {X 0,Y 495.443,Z 273.084,A -85,B 0,C 180,E1 -6273.913,E2 -6273.913} C_VEL
LIN {X 0,Y 495.406,Z 274.613,A -85,B 0,C 180,E1 -6275.899,E2 -6275.899} C_VEL
LIN {X 0,Y 499.818,Z 289.637,A -85,B 0,C 180,E1 -6276.436,E2 -6276.436} C_VEL
LIN {X 0,Y 499.943,Z 293.218,A -85,B 0,C 180,E1 -6276.55,E2 -6276.55} C_VEL
LIN {X 0,Y 499.575,Z 307.856,A -85,B 0,C 180,E1 -6277.076,E2 -6277.076} C_VEL
LIN {X 0,Y 499.054,Z 322.382,A -85,B 0,C 180,E1 -6277.761,E2 -6277.761} C_VEL
LIN {X 0,Y 498.555,Z 335.502,A -85,B 0,C 180,E1 -6278.541,E2 -6278.541} C_VEL
LIN {X 0,Y 498.074,Z 348.081,A -85,B 0,C 180,E1 -6279.452,E2 -6279.452} C_VEL
LIN {X 0,Y 497.471,Z 360.169,A -85,B 0,C 180,E1 -6280.503,E2 -6280.503} C_VEL
LIN {X 0,Y 496.956,Z 372.003,A -85,B 0,C 180,E1 -6281.743,E2 -6281.743} C_VEL
LIN {X 0,Y 496.416,Z 382.986,A -85,B 0,C 180,E1 -6283.129,E2 -6283.129} C_VEL
LIN {X 0,Y 495.952,Z 392.735,A -85,B 0,C 180,E1 -6284.62,E2 -6284.62} C_VEL
LIN {X 0,Y 495.672,Z 400.449,A -85,B 0,C 180,E1 -6286.052,E2 -6286.052} C_VEL
LIN {X 0,Y 495.408,Z 407.73,A -85,B 0,C 180,E1 -6287.714,E2 -6287.714} C_VEL
LIN {X 0,Y 495.224,Z 413.416,A -85,B 0,C 180,E1 -6289.369,E2 -6289.369} C_VEL
LIN {X 0,Y 495.062,Z 417.697,A -85,B 0,C 180,E1 -6291.016,E2 -6291.016} C_VEL
LIN {X 0,Y 495.068,Z 420.68,A -85,B 0,C 180,E1 -6292.66,E2 -6292.66} C_VEL
LIN {X 0,Y 495.077,Z 422.471,A -85,B 0,C 180,E1 -6294.297,E2 -6294.297} C_VEL
LIN {X 0,Y 495.074,Z 423.091,A -85,B 0,C 180,E1 -6295.93,E2 -6295.93} C_VEL
LIN {X 0,Y 495.049,Z 422.559,A -85,B 0,C 180,E1 -6297.559,E2 -6297.559} C_VEL
LIN {X 0,Y 494.917,Z 420.898,A -85,B 0,C 180,E1 -6299.187,E2 -6299.187} C_VEL
LIN {X 0,Y 494.945,Z 418.081,A -85,B 0,C 180,E1 -6300.814,E2 -6300.814} C_VEL
LIN {X 0,Y 495.114,Z 414.004,A -85,B 0,C 180,E1 -6302.441,E2 -6302.441} C_VEL
LIN {X 0,Y 495.414,Z 408.622,A -85,B 0,C 180,E1 -6304.068,E2 -6304.068} C_VEL
LIN {X 0,Y 495.537,Z 401.773,A -85,B 0,C 180,E1 -6305.698,E2 -6305.698} C_VEL
LIN {X 0,Y 495.902,Z 393.82,A -85,B 0,C 180,E1 -6307.226,E2 -6307.226} C_VEL
LIN {X 0,Y 496.348,Z 384.131,A -85,B 0,C 180,E1 -6308.755,E2 -6308.755} C_VEL
LIN {X 0,Y 496.835,Z 374.87,A -85,B 0,C 180,E1 -6309.979,E2 -6309.979} C_VEL
LIN {X 0,Y 497.419,Z 362.916,A -85,B 0,C 180,E1 -6311.306,E2 -6311.306} C_VEL
LIN {X 0,Y 498.007,Z 350.732,A -85,B 0,C 180,E1 -6312.428,E2 -6312.428} C_VEL
LIN {X 0,Y 498.522,Z 337.182,A -85,B 0,C 180,E1 -6313.464,E2 -6313.464} C_VEL
LIN {X 0,Y 499.209,Z 322.401,A -85,B 0,C 180,E1 -6314.367,E2 -6314.367} C_VEL
LIN {X 0,Y 499.71,Z 309.066,A -85,B 0,C 180,E1 -6315.02,E2 -6315.02} C_VEL
LIN {X 0,Y 500.135,Z 293.538,A -85,B 0,C 180,E1 -6315.6,E2 -6315.6} C_VEL
LIN {X 0,Y 499.95,Z 289.397,A -85,B 0,C 180,E1 -6315.732,E2 -6315.732} C_VEL
LIN {X 0,Y 496.511,Z 276.816,A -85,B 0,C 180,E1 -6316.184,E2 -6316.184} C_VEL
LIN {X 0,Y 495.123,Z 271.966,A -85,B 0,C 180,E1 -6316.337,E2 -6316.337} C_VEL
LIN {X 0,Y 495.135,Z 269.227,A -85,B 0,C 180,E1 -6319.055,E2 -6319.055} C_VEL
LIN {X 0,Y 495.16,Z 266.619,A -85,B 0,C 180,E1 -6321.656,E2 -6321.656} C_VEL
LIN {X 0,Y 495.258,Z 263.589,A -85,B 0,C 180,E1 -6324.742,E2 -6324.742} C_VEL
LIN {X 0,Y 495.258,Z 260.467,A -85,B 0,C 180,E1 -6327.924,E2 -6327.924} C_VEL
LIN {X 0,Y 495.291,Z 258.418,A -85,B 0,C 180,E1 -6330.052,E2 -6330.052} C_VEL
LIN {X 0,Y 495.611,Z 258.379,A -85,B 0,C 180,E1 -6333.212,E2 -6333.212} C_VEL
LIN {X 0,Y 495.743,Z 258.361,A -85,B 0,C 180,E1 -6335.538,E2 -6335.538} C_VEL
LIN {X 0,Y 495.766,Z 258.358,A -85,B 0,C 180,E1 -6338.768,E2 -6338.768} C_VEL
LIN {X 0,Y 495.754,Z 258.358,A -85,B 0,C 180,E1 -6341.782,E2 -6341.782} C_VEL
LIN {X 0,Y 495.741,Z 258.359,A -85,B 0,C 180,E1 -6345.141,E2 -6345.141} C_VEL
LIN {X 0,Y 495.76,Z 258.357,A -85,B 0,C 180,E1 -6348.219,E2 -6348.219} C_VEL
LIN {X 0,Y 495.752,Z 258.356,A -85,B 0,C 180,E1 -6351.408,E2 -6351.408} C_VEL
LIN {X 0,Y 495.75,Z 258.357,A -85,B 0,C 180,E1 -6354.462,E2 -6354.462} C_VEL
LIN {X 0,Y 495.746,Z 258.357,A -85,B 0,C 180,E1 -6354.945,E2 -6354.945} C_VEL
LIN {X 0,Y 495.096,Z 258.441,A -85,B 0,C 180,E1 -6355.623,E2 -6355.623} C_VEL
LIN {X 0,Y 492.237,Z 258.798,A -85,B 0,C 180,E1 -6356.723,E2 -6356.723} C_VEL
LIN {X 0,Y 489.81,Z 259.097,A -85,B 0,C 180,E1 -6357.61,E2 -6357.61} C_VEL
LIN {X 0,Y 488.771,Z 259.228,A -85,B 0,C 180,E1 -6358.295,E2 -6358.295} C_VEL
LIN {X 0,Y 488.689,Z 259.236,A -85,B 0,C 180,E1 -6358.527,E2 -6358.527} C_VEL
LIN {X 0,Y 488.747,Z 259.231,A -85,B 0,C 180,E1 -6361.671,E2 -6361.671} C_VEL
LIN {X 0,Y 488.709,Z 259.237,A -85,B 0,C 180,E1 -6364.442,E2 -6364.442} C_VEL
LIN {X 0,Y 488.725,Z 259.234,A -85,B 0,C 180,E1 -6367.153,E2 -6367.153} C_VEL
LIN {X 0,Y 488.727,Z 259.231,A -85,B 0,C 180,E1 -6369.81,E2 -6369.81} C_VEL
LIN {X 0,Y 488.713,Z 259.235,A -85,B 0,C 180,E1 -6372.423,E2 -6372.423} C_VEL
LIN {X 0,Y 488.764,Z 259.23,A -85,B 0,C 180,E1 -6375,E2 -6375} C_VEL
LIN {X 0,Y 488.809,Z 259.224,A -85,B 0,C 180,E1 -6378.388,E2 -6378.388} C_VEL
LIN {X 0,Y 488.82,Z 259.221,A -85,B 0,C 180,E1 -6381.734,E2 -6381.734} C_VEL
LIN {X 0,Y 488.796,Z 259.221,A -85,B 0,C 180,E1 -6385.051,E2 -6385.051} C_VEL
LIN {X 0,Y 488.959,Z 259.206,A -85,B 0,C 180,E1 -6387.529,E2 -6387.529} C_VEL
LIN {X 0,Y 488.973,Z 259.203,A -85,B 0,C 180,E1 -6390,E2 -6390} C_VEL
LIN {X 0,Y 488.957,Z 259.202,A -85,B 0,C 180,E1 -6392.471,E2 -6392.471} C_VEL
LIN {X 0,Y 488.844,Z 259.218,A -85,B 0,C 180,E1 -6395.776,E2 -6395.776} C_VEL
LIN {X 0,Y 488.787,Z 259.224,A -85,B 0,C 180,E1 -6398.267,E2 -6398.267} C_VEL
LIN {X 0,Y 488.809,Z 259.222,A -85,B 0,C 180,E1 -6401.612,E2 -6401.612} C_VEL
LIN {X 0,Y 488.761,Z 259.227,A -85,B 0,C 180,E1 -6405.001,E2 -6405.001} C_VEL
LIN {X 0,Y 488.751,Z 259.231,A -85,B 0,C 180,E1 -6408.442,E2 -6408.442} C_VEL
LIN {X 0,Y 488.711,Z 259.234,A -85,B 0,C 180,E1 -6411.071,E2 -6411.071} C_VEL
LIN {X 0,Y 488.691,Z 259.236,A -85,B 0,C 180,E1 -6413.746,E2 -6413.746} C_VEL
LIN {X 0,Y 488.795,Z 259.224,A -85,B 0,C 180,E1 -6416.943,E2 -6416.943} C_VEL
LIN {X 0,Y 488.711,Z 259.233,A -85,B 0,C 180,E1 -6420.362,E2 -6420.362} C_VEL
LIN {X 0,Y 488.738,Z 259.232,A -85,B 0,C 180,E1 -6423.484,E2 -6423.484} C_VEL
LIN {X 0,Y 488.677,Z 259.236,A -85,B 0,C 180,E1 -6426.353,E2 -6426.353} C_VEL
LIN {X 0,Y 488.7,Z 259.236,A -85,B 0,C 180,E1 -6429.255,E2 -6429.255} C_VEL
LIN {X 0,Y 488.669,Z 259.239,A -85,B 0,C 180,E1 -6432.528,E2 -6432.528} C_VEL
LIN {X 0,Y 488.705,Z 259.235,A -85,B 0,C 180,E1 -6435.197,E2 -6435.197} C_VEL
LIN {X 0,Y 488.711,Z 259.233,A -85,B 0,C 180,E1 -6438.4,E2 -6438.4} C_VEL
LIN {X 0,Y 488.708,Z 259.236,A -85,B 0,C 180,E1 -6440.947,E2 -6440.947} C_VEL
LIN {X 0,Y 488.682,Z 259.239,A -85,B 0,C 180,E1 -6443.868,E2 -6443.868} C_VEL
LIN {X 0,Y 488.74,Z 259.233,A -85,B 0,C 180,E1 -6446.877,E2 -6446.877} C_VEL
LIN {X 0,Y 488.729,Z 259.233,A -85,B 0,C 180,E1 -6449.781,E2 -6449.781} C_VEL
LIN {X 0,Y 488.737,Z 259.233,A -85,B 0,C 180,E1 -6452.602,E2 -6452.602} C_VEL
LIN {X 0,Y 488.716,Z 259.233,A -85,B 0,C 180,E1 -6455.352,E2 -6455.352} C_VEL
LIN {X 0,Y 488.702,Z 259.235,A -85,B 0,C 180,E1 -6458.043,E2 -6458.043} C_VEL
LIN {X 0,Y 488.744,Z 259.231,A -85,B 0,C 180,E1 -6460.686,E2 -6460.686} C_VEL
LIN {X 0,Y 488.766,Z 259.227,A -85,B 0,C 180,E1 -6464.145,E2 -6464.145} C_VEL
LIN {X 0,Y 488.743,Z 259.228,A -85,B 0,C 180,E1 -6467.543,E2 -6467.543} C_VEL
LIN {X 0,Y 488.765,Z 259.228,A -85,B 0,C 180,E1 -6470.064,E2 -6470.064} C_VEL
LIN {X 0,Y 488.826,Z 259.221,A -85,B 0,C 180,E1 -6472.767,E2 -6472.767} C_VEL
LIN {X 0,Y 488.797,Z 259.222,A -85,B 0,C 180,E1 -6475.051,E2 -6475.051} C_VEL
LIN {X 0,Y 488.96,Z 259.205,A -85,B 0,C 180,E1 -6477.528,E2 -6477.528} C_VEL
LIN {X 0,Y 488.973,Z 259.203,A -85,B 0,C 180,E1 -6480,E2 -6480} C_VEL
LIN {X 0,Y 488.965,Z 259.202,A -85,B 0,C 180,E1 -6482.471,E2 -6482.471} C_VEL
LIN {X 0,Y 488.841,Z 259.218,A -85,B 0,C 180,E1 -6485.776,E2 -6485.776} C_VEL
LIN {X 0,Y 488.766,Z 259.227,A -85,B 0,C 180,E1 -6488.267,E2 -6488.267} C_VEL
LIN {X 0,Y 488.81,Z 259.222,A -85,B 0,C 180,E1 -6491.612,E2 -6491.612} C_VEL
LIN {X 0,Y 488.761,Z 259.226,A -85,B 0,C 180,E1 -6495,E2 -6495} C_VEL
LIN {X 0,Y 488.751,Z 259.231,A -85,B 0,C 180,E1 -6498.442,E2 -6498.442} C_VEL
LIN {X 0,Y 488.71,Z 259.234,A -85,B 0,C 180,E1 -6501.07,E2 -6501.07} C_VEL
LIN {X 0,Y 488.678,Z 259.238,A -85,B 0,C 180,E1 -6503.746,E2 -6503.746} C_VEL
LIN {X 0,Y 488.716,Z 259.234,A -85,B 0,C 180,E1 -6506.474,E2 -6506.474} C_VEL
LIN {X 0,Y 488.703,Z 259.238,A -85,B 0,C 180,E1 -6509.271,E2 -6509.271} C_VEL
LIN {X 0,Y 488.705,Z 259.238,A -85,B 0,C 180,E1 -6512.147,E2 -6512.147} C_VEL
LIN {X 0,Y 488.717,Z 259.237,A -85,B 0,C 180,E1 -6515.115,E2 -6515.115} C_VEL
LIN {X 0,Y 488.682,Z 259.237,A -85,B 0,C 180,E1 -6518.2,E2 -6518.2} C_VEL
LIN {X 0,Y 488.679,Z 259.239,A -85,B 0,C 180,E1 -6521.418,E2 -6521.418} C_VEL
LIN {X 0,Y 488.701,Z 259.376,A -85,B 0,C 180,E1 -6522.149,E2 -6522.149} C_VEL
LIN {X 0,Y 489.884,Z 265.442,A -85,B 0,C 180,E1 -6525.334,E2 -6525.334} C_VEL
LIN {X 0,Y 490.663,Z 270.193,A -85,B 0,C 180,E1 -6527.685,E2 -6527.685} C_VEL
LIN {X 0,Y 490.688,Z 274.981,A -85,B 0,C 180,E1 -6529.87,E2 -6529.87} C_VEL
LIN {X 0,Y 490.333,Z 282.251,A -85,B 0,C 180,E1 -6532.987,E2 -6532.987} C_VEL
LIN {X 0,Y 489.963,Z 289.588,A -85,B 0,C 180,E1 -6535.984,E2 -6535.984} C_VEL
LIN {X 0,Y 489.563,Z 298.544,A -85,B 0,C 180,E1 -6539.467,E2 -6539.467} C_VEL
LIN {X 0,Y 489.302,Z 305.713,A -85,B 0,C 180,E1 -6542.172,E2 -6542.172} C_VEL
LIN {X 0,Y 489.001,Z 314.645,A -85,B 0,C 180,E1 -6545.368,E2 -6545.368} C_VEL
LIN {X 0,Y 488.765,Z 323.434,A -85,B 0,C 180,E1 -6548.49,E2 -6548.49} C_VEL
LIN {X 0,Y 488.707,Z 325.397,A -85,B 0,C 180,E1 -6549.188,E2 -6549.188} C_VEL
LIN {X 0,Y 493.217,Z 343.533,A -85,B 0,C 180,E1 -6549.76,E2 -6549.76} C_VEL
LIN {X 0,Y 493.899,Z 347.234,A -85,B 0,C 180,E1 -6549.897,E2 -6549.897} C_VEL
LIN {X 0,Y 493.439,Z 361.268,A -85,B 0,C 180,E1 -6550.365,E2 -6550.365} C_VEL
LIN {X 0,Y 492.865,Z 375.801,A -85,B 0,C 180,E1 -6551.016,E2 -6551.016} C_VEL
LIN {X 0,Y 492.167,Z 389.485,A -85,B 0,C 180,E1 -6551.798,E2 -6551.798} C_VEL
LIN {X 0,Y 491.482,Z 402.767,A -85,B 0,C 180,E1 -6552.739,E2 -6552.739} C_VEL
LIN {X 0,Y 490.785,Z 414.76,A -85,B 0,C 180,E1 -6553.765,E2 -6553.765} C_VEL
LIN {X 0,Y 490.228,Z 425.3,A -85,B 0,C 180,E1 -6554.833,E2 -6554.833} C_VEL
LIN {X 0,Y 489.658,Z 435.805,A -85,B 0,C 180,E1 -6556.089,E2 -6556.089} C_VEL
LIN {X 0,Y 489.051,Z 446.038,A -85,B 0,C 180,E1 -6557.551,E2 -6557.551} C_VEL
LIN {X 0,Y 488.722,Z 454.565,A -85,B 0,C 180,E1 -6559.016,E2 -6559.016} C_VEL
LIN {X 0,Y 488.36,Z 461.645,A -85,B 0,C 180,E1 -6560.474,E2 -6560.474} C_VEL
LIN {X 0,Y 488.141,Z 468.21,A -85,B 0,C 180,E1 -6562.139,E2 -6562.139} C_VEL
LIN {X 0,Y 488.038,Z 472.582,A -85,B 0,C 180,E1 -6563.532,E2 -6563.532} C_VEL
LIN {X 0,Y 487.934,Z 476.294,A -85,B 0,C 180,E1 -6565.042,E2 -6565.042} C_VEL
LIN {X 0,Y 487.948,Z 479.192,A -85,B 0,C 180,E1 -6566.697,E2 -6566.697} C_VEL
LIN {X 0,Y 487.886,Z 480.916,A -85,B 0,C 180,E1 -6568.349,E2 -6568.349} C_VEL
LIN {X 0,Y 487.816,Z 481.5,A -85,B 0,C 180,E1 -6570,E2 -6570} C_VEL
LIN {X 0,Y 487.886,Z 480.912,A -85,B 0,C 180,E1 -6571.651,E2 -6571.651} C_VEL
LIN {X 0,Y 487.948,Z 479.185,A -85,B 0,C 180,E1 -6573.303,E2 -6573.303} C_VEL
LIN {X 0,Y 487.934,Z 476.291,A -85,B 0,C 180,E1 -6574.958,E2 -6574.958} C_VEL
LIN {X 0,Y 488.094,Z 472.16,A -85,B 0,C 180,E1 -6576.615,E2 -6576.615} C_VEL
LIN {X 0,Y 488.201,Z 466.687,A -85,B 0,C 180,E1 -6578.277,E2 -6578.277} C_VEL
LIN {X 0,Y 488.393,Z 459.727,A -85,B 0,C 180,E1 -6579.944,E2 -6579.944} C_VEL
LIN {X 0,Y 488.816,Z 452.265,A -85,B 0,C 180,E1 -6581.402,E2 -6581.402} C_VEL
LIN {X 0,Y 489.169,Z 443.29,A -85,B 0,C 180,E1 -6582.867,E2 -6582.867} C_VEL
LIN {X 0,Y 489.725,Z 434.174,A -85,B 0,C 180,E1 -6584.121,E2 -6584.121} C_VEL
LIN {X 0,Y 490.294,Z 423.377,A -85,B 0,C 180,E1 -6585.378,E2 -6585.378} C_VEL
LIN {X 0,Y 490.984,Z 411.689,A -85,B 0,C 180,E1 -6586.519,E2 -6586.519} C_VEL
LIN {X 0,Y 491.681,Z 398.679,A -85,B 0,C 180,E1 -6587.575,E2 -6587.575} C_VEL
LIN {X 0,Y 492.43,Z 384.391,A -85,B 0,C 180,E1 -6588.515,E2 -6588.515} C_VEL
LIN {X 0,Y 493.075,Z 371.355,A -85,B 0,C 180,E1 -6589.204,E2 -6589.204} C_VEL
LIN {X 0,Y 493.62,Z 355.874,A -85,B 0,C 180,E1 -6589.835,E2 -6589.835} C_VEL
LIN {X 0,Y 493.752,Z 345.913,A -85,B 0,C 180,E1 -6590.148,E2 -6590.148} C_VEL
LIN {X 0,Y 489.907,Z 330.091,A -85,B 0,C 180,E1 -6590.672,E2 -6590.672} C_VEL
LIN {X 0,Y 488.707,Z 325.398,A -85,B 0,C 180,E1 -6590.812,E2 -6590.812} C_VEL
LIN {X 0,Y 488.929,Z 317.131,A -85,B 0,C 180,E1 -6593.733,E2 -6593.733} C_VEL
LIN {X 0,Y 489.149,Z 309.115,A -85,B 0,C 180,E1 -6596.449,E2 -6596.449} C_VEL
LIN {X 0,Y 489.387,Z 299.735,A -85,B 0,C 180,E1 -6599.7,E2 -6599.7} C_VEL
LIN {X 0,Y 489.655,Z 290.605,A -85,B 0,C 180,E1 -6603.053,E2 -6603.053} C_VEL
LIN {X 0,Y 489.935,Z 283.235,A -85,B 0,C 180,E1 -6606.025,E2 -6606.025} C_VEL
LIN {X 0,Y 490.408,Z 276.639,A -85,B 0,C 180,E1 -6609.092,E2 -6609.092} C_VEL
LIN {X 0,Y 490.668,Z 272.86,A -85,B 0,C 180,E1 -6611.214,E2 -6611.214} C_VEL
LIN {X 0,Y 490.564,Z 269.838,A -85,B 0,C 180,E1 -6613.446,E2 -6613.446} C_VEL
LIN {X 0,Y 490.182,Z 267.799,A -85,B 0,C 180,E1 -6615.798,E2 -6615.798} C_VEL
LIN {X 0,Y 489.8,Z 266.853,A -85,B 0,C 180,E1 -6618.257,E2 -6618.257} C_VEL
LIN {X 0,Y 489.341,Z 266.933,A -85,B 0,C 180,E1 -6620.856,E2 -6620.856} C_VEL
LIN {X 0,Y 489.025,Z 267.904,A -85,B 0,C 180,E1 -6623.898,E2 -6623.898} C_VEL
LIN {X 0,Y 488.769,Z 269.413,A -85,B 0,C 180,E1 -6626.88,E2 -6626.88} C_VEL
LIN {X 0,Y 488.627,Z 271.181,A -85,B 0,C 180,E1 -6629.774,E2 -6629.774} C_VEL
LIN {X 0,Y 488.471,Z 273.103,A -85,B 0,C 180,E1 -6632.587,E2 -6632.587} C_VEL
LIN {X 0,Y 488.388,Z 275.545,A -85,B 0,C 180,E1 -6635.627,E2 -6635.627} C_VEL
LIN {X 0,Y 492.912,Z 290.382,A -85,B 0,C 180,E1 -6636.183,E2 -6636.183} C_VEL
LIN {X 0,Y 493.247,Z 292.575,A -85,B 0,C 180,E1 -6636.266,E2 -6636.266} C_VEL
LIN {X 0,Y 492.863,Z 307.319,A -85,B 0,C 180,E1 -6636.796,E2 -6636.796} C_VEL
LIN {X 0,Y 492.317,Z 321.099,A -85,B 0,C 180,E1 -6637.44,E2 -6637.44} C_VEL
LIN {X 0,Y 491.764,Z 335.154,A -85,B 0,C 180,E1 -6638.272,E2 -6638.272} C_VEL
LIN {X 0,Y 491.202,Z 348.715,A -85,B 0,C 180,E1 -6639.261,E2 -6639.261} C_VEL
LIN {X 0,Y 490.565,Z 360.802,A -85,B 0,C 180,E1 -6640.326,E2 -6640.326} C_VEL
LIN {X 0,Y 490.087,Z 371.487,A -85,B 0,C 180,E1 -6641.45,E2 -6641.45} C_VEL
LIN {X 0,Y 489.584,Z 381.333,A -85,B 0,C 180,E1 -6642.671,E2 -6642.671} C_VEL
LIN {X 0,Y 489.098,Z 391.303,A -85,B 0,C 180,E1 -6644.156,E2 -6644.156} C_VEL
LIN {X 0,Y 488.729,Z 399.531,A -85,B 0,C 180,E1 -6645.638,E2 -6645.638} C_VEL
LIN {X 0,Y 488.428,Z 406.268,A -85,B 0,C 180,E1 -6647.113,E2 -6647.113} C_VEL
LIN {X 0,Y 488.231,Z 412.419,A -85,B 0,C 180,E1 -6648.795,E2 -6648.795} C_VEL
LIN {X 0,Y 488.016,Z 417.091,A -85,B 0,C 180,E1 -6650.467,E2 -6650.467} C_VEL
LIN {X 0,Y 487.983,Z 419.716,A -85,B 0,C 180,E1 -6651.72,E2 -6651.72} C_VEL
LIN {X 0,Y 488.011,Z 422.318,A -85,B 0,C 180,E1 -6653.564,E2 -6653.564} C_VEL
LIN {X 0,Y 487.904,Z 423.388,A -85,B 0,C 180,E1 -6655.042,E2 -6655.042} C_VEL
LIN {X 0,Y 487.951,Z 423.442,A -85,B 0,C 180,E1 -6656.697,E2 -6656.697} C_VEL
LIN {X 0,Y 487.892,Z 422.377,A -85,B 0,C 180,E1 -6658.349,E2 -6658.349} C_VEL
LIN {X 0,Y 487.841,Z 420.164,A -85,B 0,C 180,E1 -6660,E2 -6660} C_VEL
LIN {X 0,Y 487.938,Z 416.751,A -85,B 0,C 180,E1 -6661.651,E2 -6661.651} C_VEL
LIN {X 0,Y 488.226,Z 412.052,A -85,B 0,C 180,E1 -6663.301,E2 -6663.301} C_VEL
LIN {X 0,Y 488.443,Z 405.969,A -85,B 0,C 180,E1 -6664.953,E2 -6664.953} C_VEL
LIN {X 0,Y 488.659,Z 398.323,A -85,B 0,C 180,E1 -6666.607,E2 -6666.607} C_VEL
LIN {X 0,Y 489.097,Z 390.143,A -85,B 0,C 180,E1 -6668.054,E2 -6668.054} C_VEL
LIN {X 0,Y 489.6,Z 380.318,A -85,B 0,C 180,E1 -6669.502,E2 -6669.502} C_VEL
LIN {X 0,Y 490.113,Z 370.257,A -85,B 0,C 180,E1 -6670.744,E2 -6670.744} C_VEL
LIN {X 0,Y 490.767,Z 358.303,A -85,B 0,C 180,E1 -6671.985,E2 -6671.985} C_VEL
LIN {X 0,Y 491.456,Z 345.095,A -85,B 0,C 180,E1 -6673.122,E2 -6673.122} C_VEL
LIN {X 0,Y 491.951,Z 333.327,A -85,B 0,C 180,E1 -6673.962,E2 -6673.962} C_VEL
LIN {X 0,Y 492.544,Z 319.431,A -85,B 0,C 180,E1 -6674.777,E2 -6674.777} C_VEL
LIN {X 0,Y 493.087,Z 305.386,A -85,B 0,C 180,E1 -6675.428,E2 -6675.428} C_VEL
LIN {X 0,Y 493.352,Z 291.289,A -85,B 0,C 180,E1 -6675.934,E2 -6675.934} C_VEL
LIN {X 0,Y 489.902,Z 278.722,A -85,B 0,C 180,E1 -6676.414,E2 -6676.414} C_VEL
LIN {X 0,Y 488.069,Z 272.271,A -85,B 0,C 180,E1 -6676.637,E2 -6676.637} C_VEL
LIN {X 0,Y 488.08,Z 269.553,A -85,B 0,C 180,E1 -6679.341,E2 -6679.341} C_VEL
LIN {X 0,Y 488.085,Z 266.94,A -85,B 0,C 180,E1 -6681.986,E2 -6681.986} C_VEL
LIN {X 0,Y 488.203,Z 264.06,A -85,B 0,C 180,E1 -6684.915,E2 -6684.915} C_VEL
LIN {X 0,Y 488.182,Z 261.593,A -85,B 0,C 180,E1 -6687.431,E2 -6687.431} C_VEL
LIN {X 0,Y 488.199,Z 259.8,A -85,B 0,C 180,E1 -6689.305,E2 -6689.305} C_VEL
LIN {X 0,Y 488.273,Z 259.291,A -85,B 0,C 180,E1 -6690.274,E2 -6690.274} C_VEL
LIN {X 0,Y 488.586,Z 259.254,A -85,B 0,C 180,E1 -6693.457,E2 -6693.457} C_VEL
LIN {X 0,Y 488.708,Z 259.235,A -85,B 0,C 180,E1 -6695.116,E2 -6695.116} C_VEL
LIN {X 0,Y 488.681,Z 259.238,A -85,B 0,C 180,E1 -6698.2,E2 -6698.2} C_VEL
LIN {X 0,Y 488.722,Z 259.235,A -85,B 0,C 180,E1 -6700.345,E2 -6700.345} C_VEL
LIN {X 0,Y 488.68,Z 259.236,A -85,B 0,C 180,E1 -6703.656,E2 -6703.656} C_VEL
LIN {X 0,Y 488.688,Z 259.239,A -85,B 0,C 180,E1 -6706.345,E2 -6706.345} C_VEL
LIN {X 0,Y 488.737,Z 259.23,A -85,B 0,C 180,E1 -6709.677,E2 -6709.677} C_VEL
LIN {X 0,Y 488.682,Z 259.238,A -85,B 0,C 180,E1 -6712.841,E2 -6712.841} C_VEL
LIN {X 0,Y 488.727,Z 259.232,A -85,B 0,C 180,E1 -6715.887,E2 -6715.887} C_VEL
LIN {X 0,Y 488.689,Z 259.236,A -85,B 0,C 180,E1 -6718.527,E2 -6718.527} C_VEL
LIN {X 0,Y 488.026,Z 259.32,A -85,B 0,C 180,E1 -6719.215,E2 -6719.215} C_VEL
LIN {X 0,Y 485.17,Z 259.677,A -85,B 0,C 180,E1 -6720.332,E2 -6720.332} C_VEL
LIN {X 0,Y 482.77,Z 259.976,A -85,B 0,C 180,E1 -6721.233,E2 -6721.233} C_VEL
LIN {X 0,Y 481.765,Z 260.1,A -85,B 0,C 180,E1 -6721.928,E2 -6721.928} C_VEL
LIN {X 0,Y 481.697,Z 260.108,A -85,B 0,C 180,E1 -6722.164,E2 -6722.164} C_VEL
LIN {X 0,Y 481.679,Z 260.11,A -85,B 0,C 180,E1 -6724.968,E2 -6724.968} C_VEL
LIN {X 0,Y 481.652,Z 260.115,A -85,B 0,C 180,E1 -6727.705,E2 -6727.705} C_VEL
LIN {X 0,Y 481.706,Z 260.109,A -85,B 0,C 180,E1 -6730.393,E2 -6730.393} C_VEL
LIN {X 0,Y 481.679,Z 260.11,A -85,B 0,C 180,E1 -6733.033,E2 -6733.033} C_VEL
LIN {X 0,Y 481.689,Z 260.109,A -85,B 0,C 180,E1 -6735.639,E2 -6735.639} C_VEL
LIN {X 0,Y 481.754,Z 260.104,A -85,B 0,C 180,E1 -6738.215,E2 -6738.215} C_VEL
LIN {X 0,Y 481.765,Z 260.101,A -85,B 0,C 180,E1 -6741.612,E2 -6741.612} C_VEL
LIN {X 0,Y 481.766,Z 260.097,A -85,B 0,C 180,E1 -6744.979,E2 -6744.979} C_VEL
LIN {X 0,Y 481.925,Z 260.082,A -85,B 0,C 180,E1 -6747.493,E2 -6747.493} C_VEL
LIN {X 0,Y 481.943,Z 260.078,A -85,B 0,C 180,E1 -6750,E2 -6750} C_VEL
LIN {X 0,Y 481.923,Z 260.078,A -85,B 0,C 180,E1 -6752.508,E2 -6752.508} C_VEL
LIN {X 0,Y 481.803,Z 260.095,A -85,B 0,C 180,E1 -6755.861,E2 -6755.861} C_VEL
LIN {X 0,Y 481.742,Z 260.101,A -85,B 0,C 180,E1 -6758.389,E2 -6758.389} C_VEL
LIN {X 0,Y 481.754,Z 260.101,A -85,B 0,C 180,E1 -6761.785,E2 -6761.785} C_VEL
LIN {X 0,Y 481.743,Z 260.102,A -85,B 0,C 180,E1 -6765.224,E2 -6765.224} C_VEL
LIN {X 0,Y 481.712,Z 260.107,A -85,B 0,C 180,E1 -6768.722,E2 -6768.722} C_VEL
LIN {X 0,Y 481.649,Z 260.115,A -85,B 0,C 180,E1 -6771.395,E2 -6771.395} C_VEL
LIN {X 0,Y 481.677,Z 260.11,A -85,B 0,C 180,E1 -6774.113,E2 -6774.113} C_VEL
LIN {X 0,Y 481.749,Z 260.101,A -85,B 0,C 180,E1 -6777.139,E2 -6777.139} C_VEL
LIN {X 0,Y 481.68,Z 260.109,A -85,B 0,C 180,E1 -6779.741,E2 -6779.741} C_VEL
LIN {X 0,Y 481.675,Z 260.112,A -85,B 0,C 180,E1 -6782.674,E2 -6782.674} C_VEL
LIN {X 0,Y 481.664,Z 260.114,A -85,B 0,C 180,E1 -6785.204,E2 -6785.204} C_VEL
LIN {X 0,Y 481.671,Z 260.112,A -85,B 0,C 180,E1 -6788.859,E2 -6788.859} C_VEL
LIN {X 0,Y 481.627,Z 260.115,A -85,B 0,C 180,E1 -6792.163,E2 -6792.163} C_VEL
LIN {X 0,Y 481.659,Z 260.113,A -85,B 0,C 180,E1 -6795.542,E2 -6795.542} C_VEL
LIN {X 0,Y 481.66,Z 260.115,A -85,B 0,C 180,E1 -6798.958,E2 -6798.958} C_VEL
LIN {X 0,Y 481.658,Z 260.113,A -85,B 0,C 180,E1 -6801.993,E2 -6801.993} C_VEL
LIN {X 0,Y 481.689,Z 260.11,A -85,B 0,C 180,E1 -6805.318,E2 -6805.318} C_VEL
LIN {X 0,Y 481.65,Z 260.116,A -85,B 0,C 180,E1 -6808.312,E2 -6808.312} C_VEL
LIN {X 0,Y 481.705,Z 260.109,A -85,B 0,C 180,E1 -6811.219,E2 -6811.219} C_VEL
LIN {X 0,Y 481.682,Z 260.109,A -85,B 0,C 180,E1 -6814.041,E2 -6814.041} C_VEL
LIN {X 0,Y 481.679,Z 260.111,A -85,B 0,C 180,E1 -6816.812,E2 -6816.812} C_VEL
LIN {X 0,Y 481.699,Z 260.106,A -85,B 0,C 180,E1 -6819.503,E2 -6819.503} C_VEL
LIN {X 0,Y 481.694,Z 260.111,A -85,B 0,C 180,E1 -6822.158,E2 -6822.158} C_VEL
LIN {X 0,Y 481.746,Z 260.105,A -85,B 0,C 180,E1 -6824.776,E2 -6824.776} C_VEL
LIN {X 0,Y 481.756,Z 260.103,A -85,B 0,C 180,E1 -6828.215,E2 -6828.215} C_VEL
LIN {X 0,Y 481.742,Z 260.103,A -85,B 0,C 180,E1 -6831.611,E2 -6831.611} C_VEL
LIN {X 0,Y 481.781,Z 260.101,A -85,B 0,C 180,E1 -6834.139,E2 -6834.139} C_VEL
LIN {X 0,Y 481.926,Z 260.081,A -85,B 0,C 180,E1 -6837.492,E2 -6837.492} C_VEL
LIN {X 0,Y 481.943,Z 260.079,A -85,B 0,C 180,E1 -6840,E2 -6840} C_VEL
LIN {X 0,Y 481.932,Z 260.078,A -85,B 0,C 180,E1 -6842.507,E2 -6842.507} C_VEL
LIN {X 0,Y 481.8,Z 260.096,A -85,B 0,C 180,E1 -6845.86,E2 -6845.86} C_VEL
LIN {X 0,Y 481.725,Z 260.103,A -85,B 0,C 180,E1 -6848.389,E2 -6848.389} C_VEL
LIN {X 0,Y 481.756,Z 260.101,A -85,B 0,C 180,E1 -6851.785,E2 -6851.785} C_VEL
LIN {X 0,Y 481.744,Z 260.102,A -85,B 0,C 180,E1 -6855.224,E2 -6855.224} C_VEL
LIN {X 0,Y 481.712,Z 260.107,A -85,B 0,C 180,E1 -6858.722,E2 -6858.722} C_VEL
LIN {X 0,Y 481.649,Z 260.116,A -85,B 0,C 180,E1 -6861.394,E2 -6861.394} C_VEL
LIN {X 0,Y 481.659,Z 260.113,A -85,B 0,C 180,E1 -6864.114,E2 -6864.114} C_VEL
LIN {X 0,Y 481.694,Z 260.108,A -85,B 0,C 180,E1 -6867.126,E2 -6867.126} C_VEL
LIN {X 0,Y 481.669,Z 260.111,A -85,B 0,C 180,E1 -6869.742,E2 -6869.742} C_VEL
LIN {X 0,Y 481.674,Z 260.112,A -85,B 0,C 180,E1 -6872.674,E2 -6872.674} C_VEL
LIN {X 0,Y 481.637,Z 260.116,A -85,B 0,C 180,E1 -6875.709,E2 -6875.709} C_VEL
LIN {X 0,Y 481.672,Z 260.108,A -85,B 0,C 180,E1 -6878.859,E2 -6878.859} C_VEL
LIN {X 0,Y 481.683,Z 260.239,A -85,B 0,C 180,E1 -6881.705,E2 -6881.705} C_VEL
LIN {X 0,Y 482.663,Z 265.402,A -85,B 0,C 180,E1 -6884.481,E2 -6884.481} C_VEL
LIN {X 0,Y 483.547,Z 270.171,A -85,B 0,C 180,E1 -6886.912,E2 -6886.912} C_VEL
LIN {X 0,Y 483.825,Z 274.677,A -85,B 0,C 180,E1 -6889.055,E2 -6889.055} C_VEL
LIN {X 0,Y 483.425,Z 282.198,A -85,B 0,C 180,E1 -6892.367,E2 -6892.367} C_VEL
LIN {X 0,Y 483.085,Z 288.447,A -85,B 0,C 180,E1 -6894.989,E2 -6894.989} C_VEL
LIN {X 0,Y 482.737,Z 294.93,A -85,B 0,C 180,E1 -6897.608,E2 -6897.608} C_VEL
LIN {X 0,Y 482.495,Z 301.867,A -85,B 0,C 180,E1 -6900.314,E2 -6900.314} C_VEL
LIN {X 0,Y 482.195,Z 309.353,A -85,B 0,C 180,E1 -6903.139,E2 -6903.139} C_VEL
LIN {X 0,Y 481.877,Z 318.286,A -85,B 0,C 180,E1 -6906.355,E2 -6906.355} C_VEL
LIN {X 0,Y 481.68,Z 325.409,A -85,B 0,C 180,E1 -6908.877,E2 -6908.877} C_VEL
LIN {X 0,Y 485.976,Z 342.378,A -85,B 0,C 180,E1 -6909.417,E2 -6909.417} C_VEL
LIN {X 0,Y 487.205,Z 348.87,A -85,B 0,C 180,E1 -6909.658,E2 -6909.658} C_VEL
LIN {X 0,Y 486.724,Z 363.118,A -85,B 0,C 180,E1 -6910.16,E2 -6910.16} C_VEL
LIN {X 0,Y 486.008,Z 377.823,A -85,B 0,C 180,E1 -6910.848,E2 -6910.848} C_VEL
LIN {X 0,Y 485.329,Z 391.099,A -85,B 0,C 180,E1 -6911.641,E2 -6911.641} C_VEL
LIN {X 0,Y 484.599,Z 404.089,A -85,B 0,C 180,E1 -6912.595,E2 -6912.595} C_VEL
LIN {X 0,Y 483.868,Z 415.525,A -85,B 0,C 180,E1 -6913.602,E2 -6913.602} C_VEL
LIN {X 0,Y 483.184,Z 427.145,A -85,B 0,C 180,E1 -6914.822,E2 -6914.822} C_VEL
LIN {X 0,Y 482.611,Z 437.354,A -85,B 0,C 180,E1 -6916.097,E2 -6916.097} C_VEL
LIN {X 0,Y 482.007,Z 447.077,A -85,B 0,C 180,E1 -6917.539,E2 -6917.539} C_VEL
LIN {X 0,Y 481.64,Z 455.635,A -85,B 0,C 180,E1 -6919.065,E2 -6919.065} C_VEL
LIN {X 0,Y 481.238,Z 463.405,A -85,B 0,C 180,E1 -6920.756,E2 -6920.756} C_VEL
LIN {X 0,Y 481.014,Z 469.596,A -85,B 0,C 180,E1 -6922.444,E2 -6922.444} C_VEL
LIN {X 0,Y 480.935,Z 474.385,A -85,B 0,C 180,E1 -6924.129,E2 -6924.129} C_VEL
LIN {X 0,Y 480.796,Z 477.893,A -85,B 0,C 180,E1 -6925.809,E2 -6925.809} C_VEL
LIN {X 0,Y 480.799,Z 480.197,A -85,B 0,C 180,E1 -6927.487,E2 -6927.487} C_VEL
LIN {X 0,Y 480.756,Z 481.352,A -85,B 0,C 180,E1 -6929.162,E2 -6929.162} C_VEL
LIN {X 0,Y 480.756,Z 481.35,A -85,B 0,C 180,E1 -6930.838,E2 -6930.838} C_VEL
LIN {X 0,Y 480.799,Z 480.191,A -85,B 0,C 180,E1 -6932.513,E2 -6932.513} C_VEL
LIN {X 0,Y 480.796,Z 477.887,A -85,B 0,C 180,E1 -6934.191,E2 -6934.191} C_VEL
LIN {X 0,Y 480.942,Z 474.385,A -85,B 0,C 180,E1 -6935.871,E2 -6935.871} C_VEL
LIN {X 0,Y 481.014,Z 469.599,A -85,B 0,C 180,E1 -6937.556,E2 -6937.556} C_VEL
LIN {X 0,Y 481.238,Z 463.402,A -85,B 0,C 180,E1 -6939.244,E2 -6939.244} C_VEL
LIN {X 0,Y 481.636,Z 455.628,A -85,B 0,C 180,E1 -6940.935,E2 -6940.935} C_VEL
LIN {X 0,Y 481.989,Z 447.039,A -85,B 0,C 180,E1 -6942.468,E2 -6942.468} C_VEL
LIN {X 0,Y 482.611,Z 437.352,A -85,B 0,C 180,E1 -6943.903,E2 -6943.903} C_VEL
LIN {X 0,Y 483.161,Z 427.148,A -85,B 0,C 180,E1 -6945.179,E2 -6945.179} C_VEL
LIN {X 0,Y 483.896,Z 415.597,A -85,B 0,C 180,E1 -6946.391,E2 -6946.391} C_VEL
LIN {X 0,Y 484.667,Z 402.767,A -85,B 0,C 180,E1 -6947.511,E2 -6947.511} C_VEL
LIN {X 0,Y 485.432,Z 389.472,A -85,B 0,C 180,E1 -6948.464,E2 -6948.464} C_VEL
LIN {X 0,Y 486.137,Z 375.794,A -85,B 0,C 180,E1 -6949.257,E2 -6949.257} C_VEL
LIN {X 0,Y 486.72,Z 360.664,A -85,B 0,C 180,E1 -6949.942,E2 -6949.942} C_VEL
LIN {X 0,Y 487.147,Z 347.435,A -85,B 0,C 180,E1 -6950.389,E2 -6950.389} C_VEL
LIN {X 0,Y 483.341,Z 331.834,A -85,B 0,C 180,E1 -6950.934,E2 -6950.934} C_VEL
LIN {X 0,Y 481.683,Z 325.354,A -85,B 0,C 180,E1 -6951.142,E2 -6951.142} C_VEL
LIN {X 0,Y 481.866,Z 316.567,A -85,B 0,C 180,E1 -6954.103,E2 -6954.103} C_VEL
LIN {X 0,Y 482.118,Z 308.598,A -85,B 0,C 180,E1 -6956.866,E2 -6956.866} C_VEL
LIN {X 0,Y 482.394,Z 299.285,A -85,B 0,C 180,E1 -6960.174,E2 -6960.174} C_VEL
LIN {X 0,Y 482.646,Z 291.545,A -85,B 0,C 180,E1 -6963.097,E2 -6963.097} C_VEL
LIN {X 0,Y 482.964,Z 284.266,A -85,B 0,C 180,E1 -6966.111,E2 -6966.111} C_VEL
LIN {X 0,Y 483.36,Z 278.775,A -85,B 0,C 180,E1 -6968.698,E2 -6968.698} C_VEL
LIN {X 0,Y 483.682,Z 274.793,A -85,B 0,C 180,E1 -6970.925,E2 -6970.925} C_VEL
LIN {X 0,Y 483.741,Z 272.905,A -85,B 0,C 180,E1 -6972.188,E2 -6972.188} C_VEL
LIN {X 0,Y 483.5,Z 270.539,A -85,B 0,C 180,E1 -6974.244,E2 -6974.244} C_VEL
LIN {X 0,Y 483.132,Z 268.836,A -85,B 0,C 180,E1 -6976.664,E2 -6976.664} C_VEL
LIN {X 0,Y 482.662,Z 268.213,A -85,B 0,C 180,E1 -6979.062,E2 -6979.062} C_VEL
LIN {X 0,Y 482.221,Z 268.591,A -85,B 0,C 180,E1 -6982.257,E2 -6982.257} C_VEL
LIN {X 0,Y 481.899,Z 269.778,A -85,B 0,C 180,E1 -6985.335,E2 -6985.335} C_VEL
LIN {X 0,Y 481.69,Z 271.368,A -85,B 0,C 180,E1 -6988.315,E2 -6988.315} C_VEL
LIN {X 0,Y 481.538,Z 273.187,A -85,B 0,C 180,E1 -6991.208,E2 -6991.208} C_VEL
LIN {X 0,Y 481.39,Z 275.154,A -85,B 0,C 180,E1 -6994.025,E2 -6994.025} C_VEL
LIN {X 0,Y 481.366,Z 276.111,A -85,B 0,C 180,E1 -6995.322,E2 -6995.322} C_VEL
LIN {X 0,Y 486.109,Z 291.313,A -85,B 0,C 180,E1 -6995.928,E2 -6995.928} C_VEL
LIN {X 0,Y 486.502,Z 293.813,A -85,B 0,C 180,E1 -6996.028,E2 -6996.028} C_VEL
LIN {X 0,Y 486.045,Z 309.548,A -85,B 0,C 180,E1 -6996.618,E2 -6996.618} C_VEL
LIN {X 0,Y 485.462,Z 323.971,A -85,B 0,C 180,E1 -6997.329,E2 -6997.329} C_VEL
LIN {X 0,Y 484.855,Z 338.12,A -85,B 0,C 180,E1 -6998.209,E2 -6998.209} C_VEL
LIN {X 0,Y 484.268,Z 350.728,A -85,B 0,C 180,E1 -6999.172,E2 -6999.172} C_VEL
LIN {X 0,Y 483.628,Z 362.532,A -85,B 0,C 180,E1 -7000.253,E2 -7000.253} C_VEL
LIN {X 0,Y 483.137,Z 372.555,A -85,B 0,C 180,E1 -7001.336,E2 -7001.336} C_VEL
LIN {X 0,Y 482.581,Z 382.724,A -85,B 0,C 180,E1 -7002.63,E2 -7002.63} C_VEL
LIN {X 0,Y 482.151,Z 391.304,A -85,B 0,C 180,E1 -7003.922,E2 -7003.922} C_VEL
LIN {X 0,Y 481.745,Z 399.616,A -85,B 0,C 180,E1 -7005.425,E2 -7005.425} C_VEL
LIN {X 0,Y 481.403,Z 406.418,A -85,B 0,C 180,E1 -7006.922,E2 -7006.922} C_VEL
LIN {X 0,Y 481.18,Z 412.658,A -85,B 0,C 180,E1 -7008.628,E2 -7008.628} C_VEL
LIN {X 0,Y 480.972,Z 417.403,A -85,B 0,C 180,E1 -7010.326,E2 -7010.326} C_VEL
LIN {X 0,Y 480.916,Z 420.09,A -85,B 0,C 180,E1 -7011.597,E2 -7011.597} C_VEL
LIN {X 0,Y 480.944,Z 422.571,A -85,B 0,C 180,E1 -7013.287,E2 -7013.287} C_VEL
LIN {X 0,Y 480.837,Z 423.831,A -85,B 0,C 180,E1 -7014.969,E2 -7014.969} C_VEL
LIN {X 0,Y 480.881,Z 423.926,A -85,B 0,C 180,E1 -7016.649,E2 -7016.649} C_VEL
LIN {X 0,Y 480.825,Z 422.886,A -85,B 0,C 180,E1 -7018.325,E2 -7018.325} C_VEL
LIN {X 0,Y 480.764,Z 420.698,A -85,B 0,C 180,E1 -7020,E2 -7020} C_VEL
LIN {X 0,Y 480.87,Z 417.301,A -85,B 0,C 180,E1 -7021.675,E2 -7021.675} C_VEL
LIN {X 0,Y 481.178,Z 412.614,A -85,B 0,C 180,E1 -7023.35,E2 -7023.35} C_VEL
LIN {X 0,Y 481.404,Z 406.54,A -85,B 0,C 180,E1 -7025.025,E2 -7025.025} C_VEL
LIN {X 0,Y 481.642,Z 398.911,A -85,B 0,C 180,E1 -7026.704,E2 -7026.704} C_VEL
LIN {X 0,Y 482.114,Z 390.733,A -85,B 0,C 180,E1 -7028.171,E2 -7028.171} C_VEL
LIN {X 0,Y 482.631,Z 380.928,A -85,B 0,C 180,E1 -7029.64,E2 -7029.64} C_VEL
LIN {X 0,Y 483.184,Z 370.891,A -85,B 0,C 180,E1 -7030.9,E2 -7030.9} C_VEL
LIN {X 0,Y 483.873,Z 358.972,A -85,B 0,C 180,E1 -7032.158,E2 -7032.158} C_VEL
LIN {X 0,Y 484.597,Z 345.817,A -85,B 0,C 180,E1 -7033.311,E2 -7033.311} C_VEL
LIN {X 0,Y 485.13,Z 334.157,A -85,B 0,C 180,E1 -7034.16,E2 -7034.16} C_VEL
LIN {X 0,Y 485.746,Z 320.355,A -85,B 0,C 180,E1 -7034.989,E2 -7034.989} C_VEL
LIN {X 0,Y 486.35,Z 305.347,A -85,B 0,C 180,E1 -7035.697,E2 -7035.697} C_VEL
LIN {X 0,Y 486.529,Z 292.178,A -85,B 0,C 180,E1 -7036.182,E2 -7036.182} C_VEL
LIN {X 0,Y 482.703,Z 278.611,A -85,B 0,C 180,E1 -7036.715,E2 -7036.715} C_VEL
LIN {X 0,Y 481,Z 272.622,A -85,B 0,C 180,E1 -7036.916,E2 -7036.916} C_VEL
LIN {X 0,Y 481.003,Z 269.921,A -85,B 0,C 180,E1 -7039.637,E2 -7039.637} C_VEL
LIN {X 0,Y 481.08,Z 266.572,A -85,B 0,C 180,E1 -7043.021,E2 -7043.021} C_VEL
LIN {X 0,Y 481.119,Z 263.685,A -85,B 0,C 180,E1 -7045.991,E2 -7045.991} C_VEL
LIN {X 0,Y 481.132,Z 260.939,A -85,B 0,C 180,E1 -7048.819,E2 -7048.819} C_VEL
LIN {X 0,Y 481.142,Z 260.18,A -85,B 0,C 180,E1 -7049.778,E2 -7049.778} C_VEL
LIN {X 0,Y 481.459,Z 260.142,A -85,B 0,C 180,E1 -7052.691,E2 -7052.691} C_VEL
LIN {X 0,Y 481.654,Z 260.114,A -85,B 0,C 180,E1 -7055.202,E2 -7055.202} C_VEL
LIN {X 0,Y 481.654,Z 260.112,A -85,B 0,C 180,E1 -7058.007,E2 -7058.007} C_VEL
LIN {X 0,Y 481.652,Z 260.114,A -85,B 0,C 180,E1 -7061.043,E2 -7061.043} C_VEL
LIN {X 0,Y 481.657,Z 260.113,A -85,B 0,C 180,E1 -7064.458,E2 -7064.458} C_VEL
LIN {X 0,Y 481.651,Z 260.115,A -85,B 0,C 180,E1 -7067.839,E2 -7067.839} C_VEL
LIN {X 0,Y 481.664,Z 260.114,A -85,B 0,C 180,E1 -7070.654,E2 -7070.654} C_VEL
LIN {X 0,Y 481.631,Z 260.117,A -85,B 0,C 180,E1 -7073.376,E2 -7073.376} C_VEL
LIN {X 0,Y 481.68,Z 260.11,A -85,B 0,C 180,E1 -7076.327,E2 -7076.327} C_VEL
LIN {X 0,Y 481.654,Z 260.113,A -85,B 0,C 180,E1 -7079.417,E2 -7079.417} C_VEL
LIN {X 0,Y 481.697,Z 260.108,A -85,B 0,C 180,E1 -7082.164,E2 -7082.164} C_VEL
LIN {X 0,Y 481.064,Z 260.19,A -85,B 0,C 180,E1 -7082.862,E2 -7082.862} C_VEL
LIN {X 0,Y 478.207,Z 260.545,A -85,B 0,C 180,E1 -7083.996,E2 -7083.996} C_VEL
LIN {X 0,Y 475.761,Z 260.847,A -85,B 0,C 180,E1 -7084.91,E2 -7084.91} C_VEL
LIN {X 0,Y 474.699,Z 260.979,A -85,B 0,C 180,E1 -7085.616,E2 -7085.616} C_VEL
LIN {X 0,Y 474.608,Z 260.989,A -85,B 0,C 180,E1 -7085.855,E2 -7085.855} C_VEL
LIN {X 0,Y 474.674,Z 260.983,A -85,B 0,C 180,E1 -7089.185,E2 -7089.185} C_VEL
LIN {X 0,Y 474.647,Z 260.986,A -85,B 0,C 180,E1 -7091.884,E2 -7091.884} C_VEL
LIN {X 0,Y 474.703,Z 260.98,A -85,B 0,C 180,E1 -7094.544,E2 -7094.544} C_VEL
LIN {X 0,Y 474.708,Z 260.98,A -85,B 0,C 180,E1 -7098.038,E2 -7098.038} C_VEL
LIN {X 0,Y 474.73,Z 260.978,A -85,B 0,C 180,E1 -7101.486,E2 -7101.486} C_VEL
LIN {X 0,Y 474.736,Z 260.973,A -85,B 0,C 180,E1 -7104.904,E2 -7104.904} C_VEL
LIN {X 0,Y 474.89,Z 260.958,A -85,B 0,C 180,E1 -7107.455,E2 -7107.455} C_VEL
LIN {X 0,Y 474.913,Z 260.954,A -85,B 0,C 180,E1 -7110,E2 -7110} C_VEL
LIN {X 0,Y 474.889,Z 260.955,A -85,B 0,C 180,E1 -7112.545,E2 -7112.545} C_VEL
LIN {X 0,Y 474.764,Z 260.972,A -85,B 0,C 180,E1 -7115.948,E2 -7115.948} C_VEL
LIN {X 0,Y 474.714,Z 260.976,A -85,B 0,C 180,E1 -7118.514,E2 -7118.514} C_VEL
LIN {X 0,Y 474.708,Z 260.979,A -85,B 0,C 180,E1 -7121.962,E2 -7121.962} C_VEL
LIN {X 0,Y 474.702,Z 260.981,A -85,B 0,C 180,E1 -7125.456,E2 -7125.456} C_VEL
LIN {X 0,Y 474.667,Z 260.985,A -85,B 0,C 180,E1 -7129.01,E2 -7129.01} C_VEL
LIN {X 0,Y 474.592,Z 260.995,A -85,B 0,C 180,E1 -7131.729,E2 -7131.729} C_VEL
LIN {X 0,Y 474.66,Z 260.985,A -85,B 0,C 180,E1 -7134.493,E2 -7134.493} C_VEL
LIN {X 0,Y 474.684,Z 260.982,A -85,B 0,C 180,E1 -7137.334,E2 -7137.334} C_VEL
LIN {X 0,Y 474.606,Z 260.993,A -85,B 0,C 180,E1 -7140.81,E2 -7140.81} C_VEL
LIN {X 0,Y 474.641,Z 260.988,A -85,B 0,C 180,E1 -7143.984,E2 -7143.984} C_VEL
LIN {X 0,Y 474.57,Z 260.998,A -85,B 0,C 180,E1 -7146.898,E2 -7146.898} C_VEL
LIN {X 0,Y 474.609,Z 260.993,A -85,B 0,C 180,E1 -7149.644,E2 -7149.644} C_VEL
LIN {X 0,Y 474.577,Z 260.998,A -85,B 0,C 180,E1 -7152.939,E2 -7152.939} C_VEL
LIN {X 0,Y 474.61,Z 260.992,A -85,B 0,C 180,E1 -7155.895,E2 -7155.895} C_VEL
LIN {X 0,Y 474.632,Z 260.992,A -85,B 0,C 180,E1 -7159.041,E2 -7159.041} C_VEL
LIN {X 0,Y 474.614,Z 260.991,A -85,B 0,C 180,E1 -7161.704,E2 -7161.704} C_VEL
LIN {X 0,Y 474.627,Z 260.989,A -85,B 0,C 180,E1 -7164.726,E2 -7164.726} C_VEL
LIN {X 0,Y 474.639,Z 260.986,A -85,B 0,C 180,E1 -7167.788,E2 -7167.788} C_VEL
LIN {X 0,Y 474.629,Z 260.99,A -85,B 0,C 180,E1 -7170.885,E2 -7170.885} C_VEL
LIN {X 0,Y 474.635,Z 260.985,A -85,B 0,C 180,E1 -7173.627,E2 -7173.627} C_VEL
LIN {X 0,Y 474.639,Z 260.987,A -85,B 0,C 180,E1 -7176.642,E2 -7176.642} C_VEL
LIN {X 0,Y 474.657,Z 260.985,A -85,B 0,C 180,E1 -7180.089,E2 -7180.089} C_VEL
LIN {X 0,Y 474.64,Z 260.987,A -85,B 0,C 180,E1 -7182.774,E2 -7182.774} C_VEL
LIN {X 0,Y 474.647,Z 260.986,A -85,B 0,C 180,E1 -7185.421,E2 -7185.421} C_VEL
LIN {X 0,Y 474.71,Z 260.981,A -85,B 0,C 180,E1 -7188.037,E2 -7188.037} C_VEL
LIN {X 0,Y 474.714,Z 260.979,A -85,B 0,C 180,E1 -7191.486,E2 -7191.486} C_VEL
LIN {X 0,Y 474.744,Z 260.977,A -85,B 0,C 180,E1 -7194.052,E2 -7194.052} C_VEL
LIN {X 0,Y 474.892,Z 260.958,A -85,B 0,C 180,E1 -7197.455,E2 -7197.455} C_VEL
LIN {X 0,Y 474.913,Z 260.955,A -85,B 0,C 180,E1 -7200,E2 -7200} C_VEL
LIN {X 0,Y 474.898,Z 260.954,A -85,B 0,C 180,E1 -7202.544,E2 -7202.544} C_VEL
LIN {X 0,Y 474.76,Z 260.973,A -85,B 0,C 180,E1 -7205.948,E2 -7205.948} C_VEL
LIN {X 0,Y 474.701,Z 260.978,A -85,B 0,C 180,E1 -7208.514,E2 -7208.514} C_VEL
LIN {X 0,Y 474.709,Z 260.979,A -85,B 0,C 180,E1 -7211.962,E2 -7211.962} C_VEL
LIN {X 0,Y 474.703,Z 260.982,A -85,B 0,C 180,E1 -7215.455,E2 -7215.455} C_VEL
LIN {X 0,Y 474.667,Z 260.984,A -85,B 0,C 180,E1 -7219.01,E2 -7219.01} C_VEL
LIN {X 0,Y 474.592,Z 260.994,A -85,B 0,C 180,E1 -7221.729,E2 -7221.729} C_VEL
LIN {X 0,Y 474.639,Z 260.988,A -85,B 0,C 180,E1 -7224.494,E2 -7224.494} C_VEL
LIN {X 0,Y 474.64,Z 260.988,A -85,B 0,C 180,E1 -7227.324,E2 -7227.324} C_VEL
LIN {X 0,Y 474.6,Z 260.992,A -85,B 0,C 180,E1 -7230.23,E2 -7230.23} C_VEL
LIN {X 0,Y 474.637,Z 260.988,A -85,B 0,C 180,E1 -7233.22,E2 -7233.22} C_VEL
LIN {X 0,Y 474.59,Z 260.993,A -85,B 0,C 180,E1 -7236.323,E2 -7236.323} C_VEL
LIN {X 0,Y 474.627,Z 260.988,A -85,B 0,C 180,E1 -7239.547,E2 -7239.547} C_VEL
LIN {X 0,Y 474.612,Z 261.037,A -85,B 0,C 180,E1 -7241.219,E2 -7241.219} C_VEL
LIN {X 0,Y 475.889,Z 267.731,A -85,B 0,C 180,E1 -7244.856,E2 -7244.856} C_VEL
LIN {X 0,Y 476.733,Z 272.898,A -85,B 0,C 180,E1 -7247.485,E2 -7247.485} C_VEL
LIN {X 0,Y 476.82,Z 277.308,A -85,B 0,C 180,E1 -7249.569,E2 -7249.569} C_VEL
LIN {X 0,Y 476.417,Z 284.591,A -85,B 0,C 180,E1 -7252.806,E2 -7252.806} C_VEL
LIN {X 0,Y 475.971,Z 291.865,A -85,B 0,C 180,E1 -7255.868,E2 -7255.868} C_VEL
LIN {X 0,Y 475.582,Z 299.611,A -85,B 0,C 180,E1 -7258.993,E2 -7258.993} C_VEL
LIN {X 0,Y 475.305,Z 306.703,A -85,B 0,C 180,E1 -7261.76,E2 -7261.76} C_VEL
LIN {X 0,Y 474.981,Z 314.277,A -85,B 0,C 180,E1 -7264.59,E2 -7264.59} C_VEL
LIN {X 0,Y 474.703,Z 323.192,A -85,B 0,C 180,E1 -7267.819,E2 -7267.819} C_VEL
LIN {X 0,Y 474.647,Z 325.176,A -85,B 0,C 180,E1 -7268.53,E2 -7268.53} C_VEL
LIN {X 0,Y 479.43,Z 344.135,A -85,B 0,C 180,E1 -7269.169,E2 -7269.169} C_VEL
LIN {X 0,Y 480.538,Z 349.608,A -85,B 0,C 180,E1 -7269.385,E2 -7269.385} C_VEL
LIN {X 0,Y 479.934,Z 364.822,A -85,B 0,C 180,E1 -7269.94,E2 -7269.94} C_VEL
LIN {X 0,Y 479.24,Z 378.832,A -85,B 0,C 180,E1 -7270.622,E2 -7270.622} C_VEL
LIN {X 0,Y 478.487,Z 392.714,A -85,B 0,C 180,E1 -7271.48,E2 -7271.48} C_VEL
LIN {X 0,Y 477.71,Z 405.411,A -85,B 0,C 180,E1 -7272.447,E2 -7272.447} C_VEL
LIN {X 0,Y 476.9,Z 417.821,A -85,B 0,C 180,E1 -7273.585,E2 -7273.585} C_VEL
LIN {X 0,Y 476.171,Z 428.991,A -85,B 0,C 180,E1 -7274.812,E2 -7274.812} C_VEL
LIN {X 0,Y 475.557,Z 438.901,A -85,B 0,C 180,E1 -7276.104,E2 -7276.104} C_VEL
LIN {X 0,Y 474.9,Z 448.655,A -85,B 0,C 180,E1 -7277.614,E2 -7277.614} C_VEL
LIN {X 0,Y 474.576,Z 456.704,A -85,B 0,C 180,E1 -7279.116,E2 -7279.116} C_VEL
LIN {X 0,Y 474.192,Z 463.403,A -85,B 0,C 180,E1 -7280.617,E2 -7280.617} C_VEL
LIN {X 0,Y 473.959,Z 469.594,A -85,B 0,C 180,E1 -7282.331,E2 -7282.331} C_VEL
LIN {X 0,Y 473.842,Z 474.384,A -85,B 0,C 180,E1 -7284.041,E2 -7284.041} C_VEL
LIN {X 0,Y 473.706,Z 477.893,A -85,B 0,C 180,E1 -7285.746,E2 -7285.746} C_VEL
LIN {X 0,Y 473.718,Z 480.197,A -85,B 0,C 180,E1 -7287.449,E2 -7287.449} C_VEL
LIN {X 0,Y 473.684,Z 481.352,A -85,B 0,C 180,E1 -7289.15,E2 -7289.15} C_VEL
LIN {X 0,Y 473.684,Z 481.35,A -85,B 0,C 180,E1 -7290.85,E2 -7290.85} C_VEL
LIN {X 0,Y 473.718,Z 480.191,A -85,B 0,C 180,E1 -7292.551,E2 -7292.551} C_VEL
LIN {X 0,Y 473.706,Z 477.887,A -85,B 0,C 180,E1 -7294.254,E2 -7294.254} C_VEL
LIN {X 0,Y 473.853,Z 474.384,A -85,B 0,C 180,E1 -7295.959,E2 -7295.959} C_VEL
LIN {X 0,Y 473.959,Z 469.597,A -85,B 0,C 180,E1 -7297.669,E2 -7297.669} C_VEL
LIN {X 0,Y 474.192,Z 463.401,A -85,B 0,C 180,E1 -7299.383,E2 -7299.383} C_VEL
LIN {X 0,Y 474.621,Z 455.626,A -85,B 0,C 180,E1 -7301.099,E2 -7301.099} C_VEL
LIN {X 0,Y 474.958,Z 447.885,A -85,B 0,C 180,E1 -7302.514,E2 -7302.514} C_VEL
LIN {X 0,Y 475.556,Z 438.913,A -85,B 0,C 180,E1 -7303.895,E2 -7303.895} C_VEL
LIN {X 0,Y 476.151,Z 429.01,A -85,B 0,C 180,E1 -7305.188,E2 -7305.188} C_VEL
LIN {X 0,Y 476.928,Z 417.844,A -85,B 0,C 180,E1 -7306.414,E2 -7306.414} C_VEL
LIN {X 0,Y 477.709,Z 405.447,A -85,B 0,C 180,E1 -7307.553,E2 -7307.553} C_VEL
LIN {X 0,Y 478.497,Z 392.734,A -85,B 0,C 180,E1 -7308.519,E2 -7308.519} C_VEL
LIN {X 0,Y 479.248,Z 378.866,A -85,B 0,C 180,E1 -7309.377,E2 -7309.377} C_VEL
LIN {X 0,Y 479.984,Z 363.733,A -85,B 0,C 180,E1 -7310.107,E2 -7310.107} C_VEL
LIN {X 0,Y 480.366,Z 348.394,A -85,B 0,C 180,E1 -7310.661,E2 -7310.661} C_VEL
LIN {X 0,Y 476.433,Z 332.036,A -85,B 0,C 180,E1 -7311.254,E2 -7311.254} C_VEL
LIN {X 0,Y 474.629,Z 324.776,A -85,B 0,C 180,E1 -7311.487,E2 -7311.487} C_VEL
LIN {X 0,Y 474.872,Z 314.713,A -85,B 0,C 180,E1 -7314.948,E2 -7314.948} C_VEL
LIN {X 0,Y 475.131,Z 306.664,A -85,B 0,C 180,E1 -7317.796,E2 -7317.796} C_VEL
LIN {X 0,Y 475.349,Z 299.075,A -85,B 0,C 180,E1 -7320.575,E2 -7320.575} C_VEL
LIN {X 0,Y 475.628,Z 291.249,A -85,B 0,C 180,E1 -7323.65,E2 -7323.65} C_VEL
LIN {X 0,Y 476.057,Z 284.269,A -85,B 0,C 180,E1 -7326.671,E2 -7326.671} C_VEL
LIN {X 0,Y 476.49,Z 278.904,A -85,B 0,C 180,E1 -7329.363,E2 -7329.363} C_VEL
LIN {X 0,Y 476.779,Z 275.278,A -85,B 0,C 180,E1 -7331.554,E2 -7331.554} C_VEL
LIN {X 0,Y 476.638,Z 272.559,A -85,B 0,C 180,E1 -7333.739,E2 -7333.739} C_VEL
LIN {X 0,Y 476.249,Z 270.521,A -85,B 0,C 180,E1 -7336.311,E2 -7336.311} C_VEL
LIN {X 0,Y 475.874,Z 269.759,A -85,B 0,C 180,E1 -7338.349,E2 -7338.349} C_VEL
LIN {X 0,Y 475.463,Z 269.633,A -85,B 0,C 180,E1 -7340.536,E2 -7340.536} C_VEL
LIN {X 0,Y 475.065,Z 270.351,A -85,B 0,C 180,E1 -7343.719,E2 -7343.719} C_VEL
LIN {X 0,Y 474.773,Z 271.687,A -85,B 0,C 180,E1 -7346.79,E2 -7346.79} C_VEL
LIN {X 0,Y 474.59,Z 273.352,A -85,B 0,C 180,E1 -7349.769,E2 -7349.769} C_VEL
LIN {X 0,Y 474.439,Z 275.264,A -85,B 0,C 180,E1 -7352.723,E2 -7352.723} C_VEL
LIN {X 0,Y 474.363,Z 276.871,A -85,B 0,C 180,E1 -7355.004,E2 -7355.004} C_VEL
LIN {X 0,Y 479.515,Z 293.066,A -85,B 0,C 180,E1 -7355.693,E2 -7355.693} C_VEL
LIN {X 0,Y 479.795,Z 295.441,A -85,B 0,C 180,E1 -7355.786,E2 -7355.786} C_VEL
LIN {X 0,Y 479.31,Z 310.484,A -85,B 0,C 180,E1 -7356.371,E2 -7356.371} C_VEL
LIN {X 0,Y 478.699,Z 324.949,A -85,B 0,C 180,E1 -7357.104,E2 -7357.104} C_VEL
LIN {X 0,Y 478.059,Z 338.683,A -85,B 0,C 180,E1 -7357.979,E2 -7357.979} C_VEL
LIN {X 0,Y 477.415,Z 351.51,A -85,B 0,C 180,E1 -7358.972,E2 -7358.972} C_VEL
LIN {X 0,Y 476.756,Z 363.289,A -85,B 0,C 180,E1 -7360.069,E2 -7360.069} C_VEL
LIN {X 0,Y 476.156,Z 374.159,A -85,B 0,C 180,E1 -7361.275,E2 -7361.275} C_VEL
LIN {X 0,Y 475.575,Z 384.129,A -85,B 0,C 180,E1 -7362.587,E2 -7362.587} C_VEL
LIN {X 0,Y 475.069,Z 393.547,A -85,B 0,C 180,E1 -7364.069,E2 -7364.069} C_VEL
LIN {X 0,Y 474.642,Z 401.789,A -85,B 0,C 180,E1 -7365.64,E2 -7365.64} C_VEL
LIN {X 0,Y 474.34,Z 408.331,A -85,B 0,C 180,E1 -7367.159,E2 -7367.159} C_VEL
LIN {X 0,Y 474.13,Z 414.253,A -85,B 0,C 180,E1 -7368.89,E2 -7368.89} C_VEL
LIN {X 0,Y 473.901,Z 418.729,A -85,B 0,C 180,E1 -7370.612,E2 -7370.612} C_VEL
LIN {X 0,Y 473.857,Z 421.88,A -85,B 0,C 180,E1 -7372.329,E2 -7372.329} C_VEL
LIN {X 0,Y 473.865,Z 423.769,A -85,B 0,C 180,E1 -7374.041,E2 -7374.041} C_VEL
LIN {X 0,Y 473.818,Z 424.482,A -85,B 0,C 180,E1 -7375.747,E2 -7375.747} C_VEL
LIN {X 0,Y 473.858,Z 424.038,A -85,B 0,C 180,E1 -7377.45,E2 -7377.45} C_VEL
LIN {X 0,Y 473.694,Z 422.464,A -85,B 0,C 180,E1 -7379.15,E2 -7379.15} C_VEL
LIN {X 0,Y 473.718,Z 419.698,A -85,B 0,C 180,E1 -7380.85,E2 -7380.85} C_VEL
LIN {X 0,Y 473.936,Z 415.682,A -85,B 0,C 180,E1 -7382.55,E2 -7382.55} C_VEL
LIN {X 0,Y 474.274,Z 410.317,A -85,B 0,C 180,E1 -7384.249,E2 -7384.249} C_VEL
LIN {X 0,Y 474.416,Z 403.513,A -85,B 0,C 180,E1 -7385.952,E2 -7385.952} C_VEL
LIN {X 0,Y 474.929,Z 395.015,A -85,B 0,C 180,E1 -7387.654,E2 -7387.654} C_VEL
LIN {X 0,Y 475.422,Z 385.97,A -85,B 0,C 180,E1 -7389.144,E2 -7389.144} C_VEL
LIN {X 0,Y 476.088,Z 375.071,A -85,B 0,C 180,E1 -7390.634,E2 -7390.634} C_VEL
LIN {X 0,Y 476.736,Z 363.886,A -85,B 0,C 180,E1 -7391.911,E2 -7391.911} C_VEL
LIN {X 0,Y 477.446,Z 351.632,A -85,B 0,C 180,E1 -7393.081,E2 -7393.081} C_VEL
LIN {X 0,Y 478.079,Z 338.264,A -85,B 0,C 180,E1 -7394.141,E2 -7394.141} C_VEL
LIN {X 0,Y 478.805,Z 325.07,A -85,B 0,C 180,E1 -7394.993,E2 -7394.993} C_VEL
LIN {X 0,Y 479.444,Z 309.958,A -85,B 0,C 180,E1 -7395.774,E2 -7395.774} C_VEL
LIN {X 0,Y 479.95,Z 294.25,A -85,B 0,C 180,E1 -7396.387,E2 -7396.387} C_VEL
LIN {X 0,Y 475.996,Z 280.043,A -85,B 0,C 180,E1 -7396.967,E2 -7396.967} C_VEL
LIN {X 0,Y 473.932,Z 272.977,A -85,B 0,C 180,E1 -7397.224,E2 -7397.224} C_VEL
LIN {X 0,Y 473.928,Z 270.264,A -85,B 0,C 180,E1 -7399.942,E2 -7399.942} C_VEL
LIN {X 0,Y 474.006,Z 267.075,A -85,B 0,C 180,E1 -7403.18,E2 -7403.18} C_VEL
LIN {X 0,Y 474.068,Z 264.866,A -85,B 0,C 180,E1 -7405.463,E2 -7405.463} C_VEL
LIN {X 0,Y 474.036,Z 262.107,A -85,B 0,C 180,E1 -7408.322,E2 -7408.322} C_VEL
LIN {X 0,Y 474.048,Z 261.19,A -85,B 0,C 180,E1 -7409.291,E2 -7409.291} C_VEL
LIN {X 0,Y 474.368,Z 261.024,A -85,B 0,C 180,E1 -7412.233,E2 -7412.233} C_VEL
LIN {X 0,Y 474.617,Z 260.992,A -85,B 0,C 180,E1 -7415.275,E2 -7415.275} C_VEL
LIN {X 0,Y 474.613,Z 260.991,A -85,B 0,C 180,E1 -7418.457,E2 -7418.457} C_VEL
LIN {X 0,Y 474.618,Z 260.99,A -85,B 0,C 180,E1 -7421.786,E2 -7421.786} C_VEL
LIN {X 0,Y 474.62,Z 260.989,A -85,B 0,C 180,E1 -7425.298,E2 -7425.298} C_VEL
LIN {X 0,Y 474.624,Z 260.99,A -85,B 0,C 180,E1 -7428.215,E2 -7428.215} C_VEL
LIN {X 0,Y 474.615,Z 260.989,A -85,B 0,C 180,E1 -7431.543,E2 -7431.543} C_VEL
LIN {X 0,Y 474.626,Z 260.989,A -85,B 0,C 180,E1 -7434.726,E2 -7434.726} C_VEL
LIN {X 0,Y 474.638,Z 260.985,A -85,B 0,C 180,E1 -7437.788,E2 -7437.788} C_VEL
LIN {X 0,Y 474.628,Z 260.989,A -85,B 0,C 180,E1 -7440.885,E2 -7440.885} C_VEL
LIN {X 0,Y 474.63,Z 260.987,A -85,B 0,C 180,E1 -7443.626,E2 -7443.626} C_VEL
LIN {X 0,Y 474.608,Z 260.989,A -85,B 0,C 180,E1 -7445.855,E2 -7445.855} C_VEL
LIN {X 0,Y 473.925,Z 261.077,A -85,B 0,C 180,E1 -7446.563,E2 -7446.563} C_VEL
LIN {X 0,Y 471.058,Z 261.435,A -85,B 0,C 180,E1 -7447.713,E2 -7447.713} C_VEL
LIN {X 0,Y 468.666,Z 261.732,A -85,B 0,C 180,E1 -7448.64,E2 -7448.64} C_VEL
LIN {X 0,Y 467.672,Z 261.855,A -85,B 0,C 180,E1 -7449.357,E2 -7449.357} C_VEL
LIN {X 0,Y 467.609,Z 261.862,A -85,B 0,C 180,E1 -7449.599,E2 -7449.599} C_VEL
LIN {X 0,Y 467.599,Z 261.865,A -85,B 0,C 180,E1 -7452.506,E2 -7452.506} C_VEL
LIN {X 0,Y 467.607,Z 261.864,A -85,B 0,C 180,E1 -7455.196,E2 -7455.196} C_VEL
LIN {X 0,Y 467.66,Z 261.856,A -85,B 0,C 180,E1 -7457.855,E2 -7457.855} C_VEL
LIN {X 0,Y 467.684,Z 261.855,A -85,B 0,C 180,E1 -7461.357,E2 -7461.357} C_VEL
LIN {X 0,Y 467.71,Z 261.851,A -85,B 0,C 180,E1 -7463.962,E2 -7463.962} C_VEL
LIN {X 0,Y 467.855,Z 261.834,A -85,B 0,C 180,E1 -7467.417,E2 -7467.417} C_VEL
LIN {X 0,Y 467.883,Z 261.83,A -85,B 0,C 180,E1 -7470,E2 -7470} C_VEL
LIN {X 0,Y 467.854,Z 261.831,A -85,B 0,C 180,E1 -7472.583,E2 -7472.583} C_VEL
LIN {X 0,Y 467.726,Z 261.849,A -85,B 0,C 180,E1 -7476.038,E2 -7476.038} C_VEL
LIN {X 0,Y 467.672,Z 261.853,A -85,B 0,C 180,E1 -7478.643,E2 -7478.643} C_VEL
LIN {X 0,Y 467.66,Z 261.858,A -85,B 0,C 180,E1 -7482.145,E2 -7482.145} C_VEL
LIN {X 0,Y 467.641,Z 261.861,A -85,B 0,C 180,E1 -7485.695,E2 -7485.695} C_VEL
LIN {X 0,Y 467.626,Z 261.861,A -85,B 0,C 180,E1 -7489.308,E2 -7489.308} C_VEL
LIN {X 0,Y 467.538,Z 261.87,A -85,B 0,C 180,E1 -7492.074,E2 -7492.074} C_VEL
LIN {X 0,Y 467.606,Z 261.865,A -85,B 0,C 180,E1 -7494.887,E2 -7494.887} C_VEL
LIN {X 0,Y 467.623,Z 261.863,A -85,B 0,C 180,E1 -7497.769,E2 -7497.769} C_VEL
LIN {X 0,Y 467.571,Z 261.87,A -85,B 0,C 180,E1 -7501.045,E2 -7501.045} C_VEL
LIN {X 0,Y 467.591,Z 261.865,A -85,B 0,C 180,E1 -7504.242,E2 -7504.242} C_VEL
LIN {X 0,Y 467.546,Z 261.872,A -85,B 0,C 180,E1 -7507.185,E2 -7507.185} C_VEL
LIN {X 0,Y 467.561,Z 261.87,A -85,B 0,C 180,E1 -7510.267,E2 -7510.267} C_VEL
LIN {X 0,Y 467.549,Z 261.869,A -85,B 0,C 180,E1 -7513.746,E2 -7513.746} C_VEL
LIN {X 0,Y 467.558,Z 261.871,A -85,B 0,C 180,E1 -7516.256,E2 -7516.256} C_VEL
LIN {X 0,Y 467.582,Z 261.867,A -85,B 0,C 180,E1 -7518.723,E2 -7518.723} C_VEL
LIN {X 0,Y 467.569,Z 261.868,A -85,B 0,C 180,E1 -7521.956,E2 -7521.956} C_VEL
LIN {X 0,Y 467.563,Z 261.871,A -85,B 0,C 180,E1 -7525.167,E2 -7525.167} C_VEL
LIN {X 0,Y 467.587,Z 261.867,A -85,B 0,C 180,E1 -7528.26,E2 -7528.26} C_VEL
LIN {X 0,Y 467.58,Z 261.868,A -85,B 0,C 180,E1 -7531.25,E2 -7531.25} C_VEL
LIN {X 0,Y 467.593,Z 261.865,A -85,B 0,C 180,E1 -7534.159,E2 -7534.159} C_VEL
LIN {X 0,Y 467.581,Z 261.868,A -85,B 0,C 180,E1 -7536.996,E2 -7536.996} C_VEL
LIN {X 0,Y 467.626,Z 261.859,A -85,B 0,C 180,E1 -7539.777,E2 -7539.777} C_VEL
LIN {X 0,Y 467.6,Z 261.864,A -85,B 0,C 180,E1 -7542.506,E2 -7542.506} C_VEL
LIN {X 0,Y 467.607,Z 261.863,A -85,B 0,C 180,E1 -7545.196,E2 -7545.196} C_VEL
LIN {X 0,Y 467.662,Z 261.857,A -85,B 0,C 180,E1 -7547.854,E2 -7547.854} C_VEL
LIN {X 0,Y 467.673,Z 261.856,A -85,B 0,C 180,E1 -7551.357,E2 -7551.357} C_VEL
LIN {X 0,Y 467.709,Z 261.852,A -85,B 0,C 180,E1 -7553.962,E2 -7553.962} C_VEL
LIN {X 0,Y 467.857,Z 261.834,A -85,B 0,C 180,E1 -7557.417,E2 -7557.417} C_VEL
LIN {X 0,Y 467.883,Z 261.831,A -85,B 0,C 180,E1 -7560,E2 -7560} C_VEL
LIN {X 0,Y 467.863,Z 261.831,A -85,B 0,C 180,E1 -7562.583,E2 -7562.583} C_VEL
LIN {X 0,Y 467.723,Z 261.851,A -85,B 0,C 180,E1 -7566.037,E2 -7566.037} C_VEL
LIN {X 0,Y 467.662,Z 261.855,A -85,B 0,C 180,E1 -7568.643,E2 -7568.643} C_VEL
LIN {X 0,Y 467.661,Z 261.859,A -85,B 0,C 180,E1 -7572.145,E2 -7572.145} C_VEL
LIN {X 0,Y 467.643,Z 261.86,A -85,B 0,C 180,E1 -7575.695,E2 -7575.695} C_VEL
LIN {X 0,Y 467.617,Z 261.863,A -85,B 0,C 180,E1 -7578.763,E2 -7578.763} C_VEL
LIN {X 0,Y 467.584,Z 261.867,A -85,B 0,C 180,E1 -7581.268,E2 -7581.268} C_VEL
LIN {X 0,Y 467.563,Z 261.869,A -85,B 0,C 180,E1 -7583.944,E2 -7583.944} C_VEL
LIN {X 0,Y 467.566,Z 261.868,A -85,B 0,C 180,E1 -7586.803,E2 -7586.803} C_VEL
LIN {X 0,Y 467.545,Z 261.87,A -85,B 0,C 180,E1 -7589.739,E2 -7589.739} C_VEL
LIN {X 0,Y 467.584,Z 261.867,A -85,B 0,C 180,E1 -7592.758,E2 -7592.758} C_VEL
LIN {X 0,Y 467.555,Z 261.869,A -85,B 0,C 180,E1 -7595.889,E2 -7595.889} C_VEL
LIN {X 0,Y 467.557,Z 261.866,A -85,B 0,C 180,E1 -7599.147,E2 -7599.147} C_VEL
LIN {X 0,Y 467.577,Z 261.949,A -85,B 0,C 180,E1 -7600.789,E2 -7600.789} C_VEL
LIN {X 0,Y 468.661,Z 267.649,A -85,B 0,C 180,E1 -7603.961,E2 -7603.961} C_VEL
